C05459=1036.892,199.559,395.178,170.238,41.811,157.916
C05460=1036.886,199.310,395.204,170.234,41.811,157.916
C05461=1036.880,199.061,395.228,170.231,41.811,157.916
C05462=1036.873,198.813,395.253,170.228,41.811,157.916
C05463=1036.868,198.564,395.277,170.225,41.811,157.916
C05464=1036.861,198.316,395.302,170.222,41.811,157.915
C05465=1036.855,198.066,395.327,170.219,41.810,157.915
C05466=1036.848,197.818,395.351,170.215,41.810,157.915
C05467=1036.843,197.570,395.376,170.212,41.810,157.915
C05468=1036.836,197.321,395.400,170.209,41.810,157.915
C05469=1036.830,197.072,395.425,170.206,41.810,157.914
C05470=1036.824,196.823,395.450,170.203,41.810,157.914
C05471=1036.817,196.575,395.474,170.199,41.810,157.914
C05472=1036.812,196.326,395.499,170.196,41.810,157.914
C05473=1036.805,196.077,395.523,170.193,41.809,157.913
C05474=1036.799,195.828,395.548,170.190,41.810,157.913
C05475=1036.793,195.580,395.572,170.187,41.810,157.913
C05476=1036.787,195.331,395.597,170.184,41.809,157.913
C05477=1036.780,195.082,395.621,170.180,41.809,157.913
C05478=1036.774,194.833,395.646,170.177,41.809,157.912
C05479=1036.768,194.585,395.670,170.174,41.809,157.912
C05480=1036.762,194.336,395.695,170.172,41.809,157.912
C05481=1036.755,194.087,395.719,170.169,41.809,157.912
C05482=1036.749,193.839,395.744,170.165,41.809,157.912
C05483=1036.743,193.590,395.768,170.162,41.808,157.911
C05484=1036.737,193.341,395.792,170.159,41.809,157.911
C05485=1036.731,193.092,395.816,170.156,41.809,157.911
C05486=1036.725,192.844,395.841,170.153,41.808,157.911
C05487=1036.718,192.595,395.865,170.150,41.808,157.910
C05488=1036.713,192.346,395.890,170.147,41.809,157.910
C05489=1036.706,192.097,395.914,170.144,41.808,157.910
C05490=1036.701,191.849,395.939,170.141,41.808,157.910
C05491=1036.694,191.600,395.963,170.138,41.808,157.910
C05492=1036.688,191.351,395.987,170.135,41.808,157.910
C05493=1036.682,191.103,396.011,170.132,41.808,157.909
C05494=1036.676,190.853,396.036,170.128,41.808,157.909
C05495=1036.670,190.606,396.060,170.125,41.808,157.909
C05496=1036.664,190.356,396.085,170.122,41.808,157.909
C05497=1036.657,190.107,396.109,170.120,41.808,157.909
C05498=1036.652,189.859,396.133,170.117,41.807,157.908
C05499=1036.645,189.610,396.157,170.114,41.807,157.908
C05500=1036.639,189.326,396.185,170.110,41.807,157.908
C05501=1036.632,189.041,396.213,170.106,41.808,157.908
C05502=1036.625,188.758,396.240,170.103,41.807,157.907
C05503=1036.618,188.473,396.268,170.100,41.807,157.907
C05504=1036.612,188.225,396.292,170.097,41.807,157.907
C05505=1036.606,187.976,396.317,170.094,41.807,157.907
C05506=1036.600,187.728,396.340,170.091,41.807,157.907
C05507=1036.594,187.478,396.365,170.088,41.807,157.906
C05508=1036.588,187.230,396.389,170.085,41.807,157.906
C05509=1036.582,186.981,396.413,170.082,41.807,157.906
C05510=1036.576,186.732,396.437,170.079,41.807,157.906
C05511=1036.570,186.483,396.461,170.075,41.807,157.906
C05512=1036.564,186.235,396.485,170.073,41.807,157.906
C05513=1036.558,185.986,396.509,170.070,41.807,157.905
C05514=1036.552,185.737,396.533,170.067,41.806,157.905
C05515=1036.546,185.488,396.557,170.064,41.806,157.905
C05516=1036.541,185.239,396.581,170.062,41.806,157.905
C05517=1036.535,184.991,396.605,170.059,41.806,157.905
C05518=1036.529,184.742,396.629,170.055,41.806,157.904
C05519=1036.523,184.493,396.653,170.052,41.806,157.904
C05520=1036.517,184.244,396.678,170.049,41.806,157.904
C05521=1036.511,183.996,396.701,170.047,41.806,157.904
C05522=1036.505,183.746,396.726,170.044,41.806,157.904
C05523=1036.499,183.498,396.750,170.041,41.806,157.903
C05524=1036.493,183.250,396.773,170.037,41.806,157.903
C05525=1036.486,183.000,396.796,170.035,41.806,157.903
C05526=1036.480,182.752,396.820,170.032,41.807,157.903
C05527=1036.474,182.503,396.844,170.029,41.806,157.903
C05528=1036.468,182.254,396.867,170.026,41.807,157.903
C05529=1036.461,182.005,396.891,170.023,41.807,157.903
C05530=1036.455,181.757,396.915,170.020,41.807,157.902
C05531=1036.449,181.507,396.938,170.018,41.807,157.902
C05532=1036.442,181.259,396.961,170.015,41.807,157.902
C05533=1036.436,181.010,396.985,170.012,41.807,157.902
C05534=1036.430,180.761,397.008,170.009,41.808,157.902
C05535=1036.423,180.512,397.032,170.005,41.808,157.902
C05536=1036.418,180.264,397.055,170.002,41.808,157.902
C05537=1036.411,180.015,397.079,170.000,41.808,157.901
C05538=1036.405,179.766,397.102,169.997,41.808,157.901
C05539=1036.399,179.517,397.126,169.994,41.809,157.901
C05540=1036.393,179.268,397.149,169.991,41.809,157.901
C05541=1036.386,179.020,397.172,169.988,41.809,157.901
C05542=1036.380,178.770,397.195,169.986,41.809,157.901
C05543=1036.374,178.522,397.219,169.983,41.810,157.901
C05544=1036.367,178.272,397.242,169.979,41.809,157.900
C05545=1036.361,178.024,397.266,169.976,41.810,157.900
C05546=1036.356,177.775,397.289,169.974,41.810,157.900
C05547=1036.349,177.526,397.313,169.971,41.810,157.900
C05548=1036.342,177.278,397.335,169.968,41.810,157.900
C05549=1036.336,177.029,397.359,169.965,41.811,157.900
C05550=1036.330,176.780,397.382,169.963,41.810,157.900
C05551=1036.324,176.531,397.406,169.960,41.811,157.899
C05552=1036.318,176.282,397.429,169.957,41.811,157.899
C05553=1036.312,176.033,397.452,169.954,41.811,157.899
C05554=1036.306,175.785,397.476,169.952,41.811,157.899
C05555=1036.299,175.535,397.499,169.949,41.812,157.899
C05556=1036.293,175.287,397.522,169.946,41.812,157.899
C05557=1036.287,175.038,397.545,169.942,41.812,157.899
C05558=1036.281,174.789,397.569,169.940,41.812,157.899
C05559=1036.275,174.540,397.592,169.937,41.813,157.898
C05560=1036.269,174.291,397.615,169.934,41.812,157.898
C05561=1036.263,174.043,397.638,169.931,41.813,157.898
C05562=1036.256,173.794,397.662,169.929,41.813,157.898
C05563=1036.250,173.545,397.685,169.926,41.813,157.898
C05564=1036.244,173.261,397.712,169.923,41.813,157.898
C05565=1036.236,172.976,397.738,169.920,41.814,157.898
C05566=1036.230,172.692,397.765,169.916,41.813,157.897
C05567=1036.222,172.406,397.791,169.913,41.814,157.897
C05568=1036.216,172.158,397.814,169.910,41.814,157.897
C05569=1036.211,171.909,397.837,169.907,41.814,157.897
C05570=1036.204,171.661,397.860,169.904,41.814,157.897
C05571=1036.198,171.411,397.883,169.902,41.815,157.897
C05572=1036.192,171.162,397.906,169.899,41.815,157.897
C05573=1036.186,170.914,397.930,169.896,41.815,157.896
C05574=1036.180,170.665,397.952,169.894,41.815,157.896
C05575=1036.174,170.415,397.976,169.891,41.816,157.896
C05576=1036.167,170.167,397.998,169.888,41.816,157.896
C05577=1036.162,169.918,398.021,169.886,41.816,157.896
C05578=1036.156,169.670,398.045,169.883,41.816,157.896
C05579=1036.150,169.421,398.068,169.879,41.817,157.896
C05580=1036.144,169.171,398.091,169.877,41.816,157.895
C05581=1036.137,168.923,398.113,169.874,41.817,157.895
C05582=1036.131,168.674,398.136,169.871,41.817,157.895
C05583=1036.126,168.425,398.159,169.869,41.817,157.895
C05584=1036.120,168.176,398.183,169.866,41.817,157.895
C05585=1036.114,167.928,398.206,169.863,41.818,157.895
C05586=1036.107,167.679,398.228,169.861,41.818,157.895
C05587=1036.101,167.429,398.251,169.858,41.818,157.895
C05588=1036.095,167.180,398.274,169.856,41.818,157.895
C05589=1036.090,166.932,398.297,169.853,41.818,157.894
C05590=1036.084,166.683,398.320,169.850,41.819,157.894
C05591=1036.077,166.434,398.343,169.847,41.818,157.894
C05592=1036.072,166.185,398.366,169.844,41.819,157.894
C05593=1036.066,165.936,398.389,169.841,41.819,157.894
C05594=1036.060,165.687,398.412,169.839,41.819,157.894
C05595=1036.055,165.439,398.434,169.836,41.819,157.894
C05596=1036.047,165.189,398.457,169.834,41.820,157.894
C05597=1036.042,164.940,398.480,169.831,41.820,157.893
C05598=1036.036,164.691,398.503,169.828,41.820,157.893
C05599=1036.030,164.443,398.526,169.826,41.820,157.893
C05600=1036.024,164.194,398.548,169.823,41.820,157.893
C05601=1036.018,163.945,398.571,169.821,41.821,157.893
C05602=1036.012,163.696,398.594,169.818,41.821,157.893
C05603=1036.007,163.447,398.617,169.814,41.821,157.893
C05604=1036.001,163.198,398.640,169.812,41.821,157.893
C05605=1035.994,162.950,398.663,169.809,41.822,157.892
C05606=1035.989,162.701,398.685,169.807,41.822,157.892
C05607=1035.983,162.452,398.708,169.804,41.822,157.892
C05608=1035.977,162.203,398.731,169.801,41.822,157.892
C05609=1035.971,161.955,398.754,169.799,41.822,157.892
C05610=1035.965,161.706,398.777,169.796,41.823,157.892
C05611=1035.960,161.456,398.799,169.794,41.822,157.892
C05612=1035.954,161.207,398.822,169.791,41.823,157.892
C05613=1035.947,160.959,398.844,169.789,41.823,157.891
C05614=1035.942,160.710,398.867,169.786,41.824,157.891
C05615=1035.936,160.461,398.890,169.784,41.823,157.891
C05616=1035.930,160.212,398.913,169.780,41.824,157.891
C05617=1035.925,159.962,398.935,169.777,41.824,157.891
C05618=1035.918,159.714,398.958,169.775,41.824,157.891
C05619=1035.912,159.465,398.980,169.772,41.825,157.891
C05620=1035.906,159.216,399.003,169.770,41.825,157.891
C05621=1035.900,158.967,399.025,169.767,41.825,157.891
C05622=1035.893,158.719,399.047,169.764,41.826,157.891
C05623=1035.888,158.470,399.070,169.762,41.826,157.890
C05624=1035.882,158.220,399.091,169.759,41.827,157.890
C05625=1035.875,157.972,399.114,169.757,41.827,157.890
C05626=1035.870,157.722,399.136,169.754,41.827,157.890
C05627=1035.863,157.474,399.158,169.751,41.828,157.890
C05628=1035.856,157.189,399.184,169.748,41.828,157.890
C05629=1035.849,156.904,399.209,169.745,41.829,157.890
C05630=1035.842,156.618,399.235,169.743,41.829,157.890
C05631=1035.835,156.333,399.260,169.740,41.829,157.890
C05632=1035.829,156.085,399.283,169.737,41.830,157.890
C05633=1035.823,155.835,399.305,169.734,41.830,157.889
C05634=1035.817,155.587,399.327,169.732,41.830,157.889
C05635=1035.811,155.337,399.349,169.729,41.831,157.889
C05636=1035.805,155.088,399.372,169.727,41.831,157.889
C05637=1035.799,154.839,399.394,169.724,41.831,157.889
C05638=1035.792,154.591,399.416,169.722,41.832,157.889
C05639=1035.786,154.342,399.439,169.719,41.832,157.889
C05640=1035.780,154.093,399.460,169.717,41.832,157.889
C05641=1035.775,153.844,399.482,169.714,41.833,157.889
C05642=1035.768,153.596,399.504,169.711,41.833,157.889
C05643=1035.763,153.346,399.526,169.709,41.834,157.889
C05644=1035.756,153.097,399.549,169.706,41.834,157.889
C05645=1035.750,152.848,399.570,169.704,41.834,157.888
C05646=1035.744,152.600,399.593,169.700,41.835,157.888
C05647=1035.738,152.350,399.614,169.698,41.835,157.888
C05648=1035.732,152.101,399.637,169.695,41.835,157.888
C05649=1035.726,151.852,399.659,169.692,41.836,157.888
C05650=1035.720,151.603,399.681,169.690,41.836,157.888
C05651=1035.713,151.355,399.703,169.687,41.837,157.888
C05652=1035.707,151.105,399.725,169.685,41.837,157.888
C05653=1035.701,150.857,399.746,169.682,41.837,157.888
C05654=1035.696,150.608,399.769,169.680,41.838,157.888
C05655=1035.689,150.359,399.790,169.677,41.839,157.888
C05656=1035.683,150.109,399.812,169.675,41.839,157.888
C05657=1035.677,149.861,399.834,169.672,41.839,157.888
C05658=1035.671,149.612,399.856,169.670,41.840,157.887
C05659=1035.664,149.362,399.878,169.667,41.840,157.887
C05660=1035.658,149.114,399.900,169.665,41.840,157.887
C05661=1035.653,148.865,399.922,169.662,41.841,157.887
C05662=1035.647,148.616,399.943,169.660,41.841,157.887
C05663=1035.641,148.367,399.965,169.657,41.841,157.887
C05664=1035.634,148.118,399.987,169.655,41.842,157.887
C05665=1035.628,147.869,400.009,169.652,41.842,157.887
C05666=1035.622,147.620,400.031,169.650,41.842,157.887
C05667=1035.616,147.371,400.052,169.647,41.843,157.887
C05668=1035.610,147.122,400.074,169.644,41.844,157.887
C05669=1035.604,146.873,400.096,169.642,41.844,157.887
C05670=1035.598,146.624,400.118,169.639,41.845,157.887
C05671=1035.592,146.375,400.139,169.637,41.845,157.886
C05672=1035.585,146.126,400.161,169.634,41.845,157.886
C05673=1035.580,145.877,400.182,169.632,41.846,157.886
C05674=1035.574,145.628,400.204,169.629,41.847,157.886
C05675=1035.567,145.379,400.225,169.627,41.847,157.886
C05676=1035.561,145.130,400.247,169.624,41.847,157.886
C05677=1035.555,144.881,400.269,169.622,41.848,157.886
C05678=1035.549,144.632,400.291,169.619,41.848,157.886
C05679=1035.543,144.383,400.312,169.617,41.849,157.886
C05680=1035.537,144.134,400.334,169.614,41.849,157.886
C05681=1035.530,143.885,400.355,169.612,41.850,157.886
C05682=1035.524,143.636,400.377,169.609,41.850,157.886
C05683=1035.518,143.388,400.398,169.607,41.850,157.886
C05684=1035.512,143.138,400.420,169.604,41.851,157.886
C05685=1035.506,142.889,400.441,169.602,41.852,157.886
C05686=1035.500,142.640,400.463,169.599,41.852,157.886
C05687=1035.494,142.391,400.484,169.597,41.852,157.886
C05688=1035.488,142.142,400.506,169.594,41.853,157.885
C05689=1035.482,141.893,400.527,169.592,41.853,157.885
C05690=1035.476,141.644,400.549,169.589,41.854,157.885
C05691=1035.469,141.395,400.570,169.587,41.854,157.885
C05692=1035.462,141.110,400.595,169.584,41.855,157.885
C05693=1035.456,140.824,400.619,169.581,41.855,157.885
C05694=1035.449,140.539,400.644,169.578,41.856,157.885
C05695=1035.442,140.254,400.669,169.576,41.857,157.885
C05696=1035.436,140.005,400.690,169.573,41.857,157.885
C05697=1035.430,139.755,400.711,169.571,41.857,157.885
C05698=1035.423,139.506,400.732,169.568,41.858,157.885
C05699=1035.418,139.258,400.753,169.566,41.858,157.885
C05700=1035.412,139.009,400.775,169.563,41.859,157.885
C05701=1035.405,138.759,400.797,169.561,41.859,157.885
C05702=1035.399,138.510,400.818,169.558,41.860,157.885
C05703=1035.393,138.262,400.839,169.556,41.860,157.885
C05704=1035.387,138.012,400.860,169.553,41.861,157.885
C05705=1035.381,137.763,400.882,169.551,41.861,157.884
C05706=1035.375,137.515,400.902,169.548,41.862,157.884
C05707=1035.368,137.266,400.924,169.546,41.862,157.884
C05708=1035.362,137.016,400.946,169.543,41.863,157.884
C05709=1035.357,136.767,400.966,169.541,41.864,157.884
C05710=1035.350,136.518,400.987,169.539,41.864,157.884
C05711=1035.344,136.269,401.009,169.536,41.865,157.884
C05712=1035.338,136.021,401.030,169.534,41.865,157.884
C05713=1035.332,135.771,401.050,169.531,41.866,157.884
C05714=1035.326,135.522,401.072,169.529,41.866,157.884
C05715=1035.320,135.273,401.093,169.526,41.867,157.884
C05716=1035.313,135.025,401.114,169.524,41.867,157.884
C05717=1035.307,134.775,401.135,169.521,41.868,157.884
C05718=1035.301,134.527,401.156,169.520,41.869,157.884
C05719=1035.295,134.277,401.178,169.516,41.869,157.884
C05720=1035.289,134.027,401.198,169.514,41.869,157.884
C05721=1035.283,133.779,401.219,169.513,41.870,157.884
C05722=1035.277,133.530,401.241,169.510,41.871,157.884
C05723=1035.271,133.280,401.262,169.508,41.871,157.884
C05724=1035.264,133.032,401.282,169.505,41.871,157.884
C05725=1035.258,132.783,401.304,169.503,41.872,157.884
C05726=1035.252,132.534,401.324,169.500,41.873,157.883
C05727=1035.246,132.285,401.346,169.498,41.873,157.883
C05728=1035.240,132.035,401.366,169.496,41.874,157.883
C05729=1035.234,131.787,401.387,169.493,41.874,157.883
C05730=1035.228,131.538,401.409,169.491,41.875,157.883
C05731=1035.222,131.289,401.429,169.488,41.875,157.883
C05732=1035.216,131.040,401.450,169.486,41.876,157.883
C05733=1035.210,130.790,401.471,169.483,41.876,157.883
C05734=1035.203,130.542,401.492,169.481,41.877,157.883
C05735=1035.197,130.292,401.512,169.478,41.878,157.883
C05736=1035.191,130.044,401.534,169.476,41.878,157.883
C05737=1035.185,129.794,401.554,169.474,41.879,157.883
C05738=1035.178,129.545,401.575,169.471,41.879,157.883
C05739=1035.172,129.296,401.596,169.469,41.880,157.883
C05740=1035.166,129.047,401.617,169.466,41.881,157.883
C05741=1035.160,128.798,401.637,169.464,41.882,157.883
C05742=1035.154,128.549,401.657,169.461,41.882,157.883
C05743=1035.147,128.300,401.678,169.459,41.882,157.883
C05744=1035.141,128.051,401.698,169.456,41.883,157.883
C05745=1035.135,127.802,401.720,169.454,41.884,157.883
C05746=1035.129,127.553,401.740,169.451,41.885,157.883
C05747=1035.122,127.303,401.760,169.449,41.885,157.883
C05748=1035.116,127.055,401.781,169.448,41.886,157.883
C05749=1035.110,126.805,401.802,169.445,41.886,157.883
C05750=1035.103,126.556,401.822,169.442,41.887,157.883
C05751=1035.097,126.308,401.843,169.440,41.888,157.883
C05752=1035.091,126.058,401.864,169.438,41.888,157.883
C05753=1035.085,125.809,401.884,169.435,41.889,157.883
C05754=1035.078,125.560,401.905,169.433,41.889,157.883
C05755=1035.073,125.311,401.925,169.431,41.890,157.883
C05756=1035.065,125.026,401.948,169.428,41.891,157.883
C05757=1035.058,124.740,401.972,169.425,41.892,157.883
C05758=1035.051,124.454,401.996,169.422,41.892,157.882
C05759=1035.044,124.169,402.020,169.420,41.893,157.883
C05760=1035.038,123.920,402.040,169.417,41.894,157.882
C05761=1035.032,123.670,402.061,169.415,41.894,157.882
C05762=1035.026,123.421,402.081,169.412,41.895,157.882
C05763=1035.019,123.173,402.102,169.410,41.895,157.882
C05764=1035.014,122.923,402.122,169.407,41.896,157.882
C05765=1035.008,122.675,402.142,169.405,41.897,157.882
C05766=1035.001,122.425,402.163,169.403,41.897,157.882
C05767=1034.995,122.177,402.183,169.400,41.898,157.882
C05768=1034.989,121.927,402.204,169.398,41.898,157.882
C05769=1034.983,121.678,402.224,169.397,41.899,157.882
C05770=1034.976,121.429,402.244,169.393,41.900,157.882
C05771=1034.970,121.180,402.264,169.392,41.900,157.882
C05772=1034.964,120.931,402.286,169.389,41.901,157.882
C05773=1034.958,120.682,402.306,169.387,41.901,157.882
C05774=1034.952,120.432,402.326,169.385,41.902,157.882
C05775=1034.946,120.183,402.347,169.382,41.903,157.882
C05776=1034.940,119.935,402.367,169.380,41.903,157.882
C05777=1034.934,119.685,402.387,169.377,41.904,157.882
C05778=1034.928,119.436,402.407,169.375,41.904,157.882
C05779=1034.922,119.187,402.429,169.373,41.905,157.882
C05780=1034.916,118.938,402.449,169.370,41.906,157.882
C05781=1034.910,118.689,402.469,169.368,41.906,157.882
C05782=1034.903,118.440,402.489,169.366,41.907,157.882
C05783=1034.898,118.191,402.510,169.363,41.907,157.882
C05784=1034.891,117.941,402.530,169.361,41.908,157.882
C05785=1034.885,117.692,402.550,169.359,41.908,157.882
C05786=1034.879,117.444,402.570,169.356,41.909,157.882
C05787=1034.873,117.194,402.591,169.354,41.910,157.882
C05788=1034.867,116.945,402.611,169.351,41.910,157.882
C05789=1034.861,116.697,402.631,169.349,41.911,157.882
C05790=1034.854,116.447,402.652,169.347,41.911,157.882
C05791=1034.849,116.198,402.672,169.344,41.912,157.881
C05792=1034.843,115.949,402.692,169.342,41.913,157.882
C05793=1034.837,115.700,402.712,169.340,41.913,157.881
C05794=1034.831,115.451,402.732,169.338,41.914,157.882
C05795=1034.825,115.202,402.753,169.335,41.914,157.881
C05796=1034.819,114.952,402.773,169.333,41.915,157.881
C05797=1034.813,114.704,402.793,169.331,41.916,157.881
C05798=1034.807,114.455,402.813,169.329,41.916,157.881
C05799=1034.800,114.205,402.834,169.327,41.916,157.881
C05800=1034.795,113.956,402.854,169.324,41.917,157.881
C05801=1034.789,113.707,402.874,169.322,41.918,157.881
C05802=1034.783,113.457,402.894,169.320,41.918,157.881
C05803=1034.777,113.208,402.914,169.317,41.919,157.881
C05804=1034.771,112.959,402.934,169.315,41.919,157.881
C05805=1034.764,112.710,402.954,169.313,41.920,157.881
C05806=1034.758,112.461,402.974,169.310,41.921,157.881
C05807=1034.752,112.212,402.994,169.308,41.922,157.881
C05808=1034.745,111.963,403.014,169.306,41.922,157.881
C05809=1034.739,111.714,403.034,169.303,41.923,157.881
C05810=1034.734,111.465,403.053,169.301,41.923,157.881
C05811=1034.727,111.215,403.074,169.299,41.924,157.881
C05812=1034.721,110.966,403.094,169.296,41.925,157.881
C05813=1034.715,110.717,403.114,169.294,41.925,157.881
C05814=1034.709,110.468,403.134,169.291,41.926,157.881
C05815=1034.703,110.218,403.153,169.289,41.927,157.881
C05816=1034.697,109.970,403.173,169.287,41.927,157.881
C05817=1034.691,109.721,403.193,169.285,41.928,157.881
C05818=1034.684,109.471,403.212,169.283,41.929,157.881
C05819=1034.678,109.222,403.232,169.281,41.929,157.881
C05820=1034.671,108.936,403.255,169.278,41.930,157.881
C05821=1034.664,108.651,403.277,169.275,41.931,157.881
C05822=1034.656,108.365,403.300,169.272,41.932,157.881
C05823=1034.649,108.079,403.323,169.270,41.933,157.881
C05824=1034.643,107.830,403.342,169.267,41.933,157.881
C05825=1034.637,107.581,403.362,169.265,41.934,157.881
C05826=1034.631,107.333,403.382,169.263,41.935,157.881
C05827=1034.625,107.083,403.402,169.260,41.936,157.881
C05828=1034.619,106.834,403.421,169.259,41.937,157.881
C05829=1034.612,106.585,403.441,169.256,41.937,157.881
C05830=1034.606,106.336,403.460,169.254,41.938,157.881
C05831=1034.600,106.086,403.480,169.252,41.938,157.881
C05832=1034.594,105.837,403.500,169.250,41.939,157.881
C05833=1034.588,105.588,403.520,169.247,41.940,157.881
C05834=1034.581,105.340,403.539,169.245,41.941,157.881
C05835=1034.575,105.089,403.559,169.243,41.941,157.881
C05836=1034.569,104.841,403.579,169.240,41.942,157.881
C05837=1034.563,104.592,403.599,169.238,41.942,157.881
C05838=1034.556,104.343,403.617,169.236,41.943,157.881
C05839=1034.550,104.094,403.637,169.233,41.944,157.881
C05840=1034.544,103.844,403.657,169.231,41.944,157.881
C05841=1034.538,103.595,403.677,169.229,41.945,157.881
C05842=1034.532,103.345,403.696,169.226,41.946,157.881
C05843=1034.526,103.097,403.715,169.224,41.947,157.881
C05844=1034.520,102.848,403.735,169.222,41.947,157.881
C05845=1034.513,102.598,403.755,169.220,41.948,157.881
C05846=1034.508,102.349,403.774,169.218,41.948,157.881
C05847=1034.501,102.100,403.793,169.216,41.949,157.881
C05848=1034.495,101.851,403.813,169.213,41.950,157.881
C05849=1034.489,101.602,403.833,169.211,41.951,157.881
C05850=1034.484,101.352,403.852,169.209,41.951,157.881
C05851=1034.476,101.103,403.872,169.206,41.952,157.881
C05852=1034.471,100.854,403.891,169.204,41.952,157.881
C05853=1034.465,100.605,403.911,169.202,41.953,157.881
C05854=1034.459,100.355,403.930,169.199,41.954,157.881
C05855=1034.453,100.107,403.950,169.197,41.955,157.881
C05856=1034.447,99.858,403.969,169.195,41.955,157.881
C05857=1034.440,99.607,403.988,169.192,41.956,157.881
C05858=1034.434,99.359,404.008,169.190,41.957,157.881
C05859=1034.428,99.109,404.027,169.188,41.957,157.881
C05860=1034.421,98.860,404.046,169.186,41.958,157.881
C05861=1034.415,98.612,404.066,169.184,41.959,157.881
C05862=1034.409,98.362,404.084,169.182,41.959,157.881
C05863=1034.402,98.113,404.103,169.179,41.961,157.881
C05864=1034.396,97.864,404.123,169.177,41.961,157.881
C05865=1034.390,97.615,404.142,169.175,41.962,157.881
C05866=1034.384,97.365,404.161,169.172,41.963,157.881
C05867=1034.377,97.117,404.180,169.170,41.963,157.881
C05868=1034.371,96.867,404.200,169.168,41.964,157.881
C05869=1034.365,96.618,404.218,169.165,41.965,157.881
C05870=1034.359,96.369,404.238,169.163,41.965,157.881
C05871=1034.352,96.120,404.257,169.161,41.966,157.881
C05872=1034.346,95.870,404.277,169.159,41.967,157.881
C05873=1034.340,95.621,404.295,169.157,41.968,157.881
C05874=1034.334,95.372,404.314,169.155,41.969,157.881
C05875=1034.327,95.123,404.334,169.152,41.969,157.881
C05876=1034.322,94.874,404.353,169.150,41.970,157.881
C05877=1034.315,94.625,404.372,169.148,41.971,157.881
C05878=1034.310,94.375,404.391,169.145,41.971,157.881
C05879=1034.303,94.127,404.410,169.143,41.972,157.881
C05880=1034.297,93.877,404.430,169.141,41.973,157.881
C05881=1034.291,93.628,404.448,169.138,41.974,157.881
C05882=1034.285,93.379,404.467,169.136,41.975,157.881
C05883=1034.279,93.129,404.486,169.134,41.975,157.881
C05884=1034.271,92.844,404.508,169.132,41.976,157.881
C05885=1034.264,92.557,404.530,169.129,41.977,157.881
C05886=1034.257,92.272,404.552,169.127,41.977,157.881
C05887=1034.250,91.986,404.574,169.124,41.978,157.881
C05888=1034.244,91.737,404.593,169.122,41.979,157.881
C05889=1034.238,91.488,404.612,169.119,41.980,157.880
C05890=1034.231,91.239,404.631,169.117,41.981,157.881
C05891=1034.226,90.990,404.650,169.115,41.981,157.880
C05892=1034.219,90.741,404.669,169.112,41.982,157.881
C05893=1034.214,90.491,404.688,169.110,41.982,157.880
C05894=1034.207,90.242,404.707,169.108,41.983,157.881
C05895=1034.201,89.993,404.726,169.106,41.984,157.881
C05896=1034.195,89.743,404.745,169.103,41.985,157.880
C05897=1034.189,89.494,404.763,169.102,41.986,157.881
C05898=1034.182,89.245,404.782,169.100,41.987,157.881
C05899=1034.176,88.996,404.801,169.097,41.987,157.880
C05900=1034.170,88.747,404.820,169.095,41.988,157.881
C05901=1034.164,88.497,404.838,169.093,41.989,157.881
C05902=1034.157,88.248,404.857,169.090,41.990,157.881
C05903=1034.151,87.999,404.876,169.088,41.990,157.881
C05904=1034.145,87.750,404.895,169.086,41.991,157.881
C05905=1034.139,87.501,404.914,169.083,41.992,157.881
C05906=1034.132,87.252,404.932,169.081,41.993,157.881
C05907=1034.126,87.002,404.951,169.079,41.993,157.881
C05908=1034.119,86.753,404.970,169.077,41.995,157.881
C05909=1034.113,86.504,404.988,169.075,41.995,157.881
C05910=1034.107,86.255,405.007,169.073,41.996,157.881
C05911=1034.101,86.005,405.025,169.070,41.997,157.881
C05912=1034.095,85.756,405.044,169.068,41.998,157.881
C05913=1034.088,85.507,405.063,169.066,41.998,157.881
C05914=1034.082,85.258,405.081,169.063,41.999,157.881
C05915=1034.075,85.009,405.100,169.061,42.000,157.881
C05916=1034.070,84.759,405.119,169.059,42.000,157.881
C05917=1034.063,84.510,405.138,169.056,42.001,157.881
C05918=1034.057,84.261,405.156,169.055,42.002,157.881
C05919=1034.051,84.011,405.174,169.053,42.003,157.881
C05920=1034.044,83.762,405.193,169.050,42.004,157.881
C05921=1034.038,83.513,405.212,169.048,42.005,157.881
C05922=1034.032,83.263,405.231,169.046,42.005,157.881
C05923=1034.026,83.014,405.250,169.043,42.006,157.881
C05924=1034.020,82.766,405.268,169.041,42.007,157.881
C05925=1034.014,82.516,405.286,169.039,42.007,157.881
C05926=1034.007,82.267,405.304,169.036,42.008,157.881
C05927=1034.001,82.018,405.323,169.034,42.009,157.881
C05928=1033.995,81.769,405.342,169.032,42.010,157.881
C05929=1033.989,81.519,405.360,169.029,42.011,157.881
C05930=1033.983,81.270,405.379,169.028,42.012,157.881
C05931=1033.976,81.020,405.398,169.026,42.012,157.881
C05932=1033.970,80.771,405.416,169.024,42.013,157.881
C05933=1033.964,80.522,405.434,169.021,42.014,157.881
C05934=1033.958,80.273,405.452,169.019,42.014,157.881
C05935=1033.952,80.024,405.471,169.017,42.015,157.881
C05936=1033.946,79.775,405.490,169.014,42.016,157.881
C05937=1033.940,79.525,405.508,169.012,42.017,157.881
C05938=1033.933,79.276,405.527,169.010,42.017,157.881
C05939=1033.927,79.027,405.546,169.007,42.018,157.881
C05940=1033.921,78.778,405.563,169.005,42.019,157.881
C05941=1033.915,78.529,405.582,169.004,42.020,157.881
C05942=1033.908,78.279,405.600,169.002,42.020,157.881
C05943=1033.902,78.030,405.618,168.999,42.021,157.881
C05944=1033.896,77.781,405.637,168.997,42.022,157.881
C05945=1033.890,77.531,405.656,168.995,42.022,157.881
C05946=1033.883,77.282,405.674,168.992,42.023,157.881
C05947=1033.878,77.033,405.692,168.990,42.024,157.881
C05948=1033.870,76.747,405.714,168.987,42.025,157.881
C05949=1033.863,76.462,405.734,168.985,42.026,157.881
C05950=1033.856,76.175,405.755,168.982,42.027,157.881
C05951=1033.849,75.889,405.776,168.979,42.028,157.881
C05952=1033.843,75.640,405.794,168.978,42.029,157.881
C05953=1033.837,75.390,405.812,168.976,42.030,157.881
C05954=1033.830,75.142,405.830,168.973,42.030,157.881
C05955=1033.824,74.893,405.848,168.971,42.031,157.881
C05956=1033.817,74.644,405.867,168.969,42.032,157.881
C05957=1033.811,74.394,405.885,168.966,42.033,157.881
C05958=1033.805,74.145,405.903,168.964,42.033,157.881
C05959=1033.799,73.895,405.921,168.962,42.034,157.881
C05960=1033.793,73.647,405.939,168.959,42.036,157.881
C05961=1033.786,73.397,405.957,168.957,42.036,157.881
C05962=1033.780,73.148,405.975,168.956,42.037,157.881
C05963=1033.774,72.898,405.993,168.953,42.038,157.881
C05964=1033.768,72.650,406.012,168.951,42.039,157.881
C05965=1033.762,72.400,406.030,168.949,42.039,157.881
C05966=1033.755,72.151,406.048,168.946,42.040,157.881
C05967=1033.749,71.901,406.066,168.944,42.041,157.881
C05968=1033.742,71.652,406.083,168.942,42.041,157.881
C05969=1033.736,71.403,406.102,168.939,42.042,157.881
C05970=1033.730,71.154,406.120,168.937,42.043,157.881
C05971=1033.724,70.904,406.138,168.936,42.044,157.881
C05972=1033.718,70.655,406.156,168.934,42.045,157.881
C05973=1033.712,70.406,406.174,168.931,42.046,157.881
C05974=1033.705,70.157,406.192,168.929,42.047,157.881
C05975=1033.699,69.907,406.210,168.927,42.047,157.881
C05976=1033.693,69.657,406.228,168.924,42.048,157.881
C05977=1033.687,69.409,406.246,168.922,42.049,157.881
C05978=1033.681,69.159,406.264,168.920,42.050,157.881
C05979=1033.674,68.910,406.281,168.917,42.050,157.881
C05980=1033.668,68.661,406.300,168.915,42.051,157.881
C05981=1033.662,68.412,406.318,168.914,42.052,157.881
C05982=1033.655,68.162,406.335,168.911,42.053,157.881
C05983=1033.649,67.913,406.354,168.909,42.054,157.881
C05984=1033.643,67.663,406.371,168.907,42.055,157.881
C05985=1033.636,67.415,406.388,168.904,42.056,157.881
C05986=1033.630,67.165,406.406,168.902,42.057,157.881
C05987=1033.624,66.916,406.425,168.900,42.057,157.881
C05988=1033.618,66.667,406.443,168.897,42.058,157.881
C05989=1033.611,66.417,406.460,168.895,42.059,157.881
C05990=1033.605,66.168,406.478,168.893,42.060,157.881
C05991=1033.599,65.919,406.495,168.890,42.060,157.881
C05992=1033.593,65.670,406.513,168.889,42.061,157.881
C05993=1033.587,65.420,406.531,168.887,42.062,157.881
C05994=1033.580,65.171,406.549,168.884,42.063,157.881
C05995=1033.574,64.921,406.566,168.882,42.064,157.881
C05996=1033.568,64.672,406.584,168.880,42.064,157.881
C05997=1033.561,64.423,406.602,168.877,42.066,157.881
C05998=1033.555,64.174,406.620,168.875,42.067,157.882
C05999=1033.548,63.924,406.637,168.873,42.067,157.882
C06000=1033.542,63.675,406.655,168.870,42.068,157.881
C06001=1033.537,63.426,406.673,168.869,42.069,157.882
C06002=1033.530,63.176,406.690,168.867,42.070,157.882
C06003=1033.523,62.927,406.707,168.864,42.071,157.882
C06004=1033.518,62.678,406.725,168.862,42.072,157.882
C06005=1033.511,62.428,406.742,168.859,42.073,157.882
C06006=1033.504,62.179,406.760,168.857,42.074,157.882
C06007=1033.498,61.929,406.778,168.855,42.075,157.882
C06008=1033.492,61.680,406.795,168.853,42.076,157.882
C06009=1033.485,61.431,406.812,168.851,42.076,157.882
C06010=1033.479,61.181,406.830,168.849,42.077,157.882
C06011=1033.472,60.933,406.847,168.846,42.078,157.882
C06012=1033.465,60.647,406.867,168.844,42.079,157.882
C06013=1033.457,60.360,406.886,168.841,42.080,157.882
C06014=1033.450,60.074,406.906,168.838,42.081,157.882
C06015=1033.443,59.789,406.927,168.835,42.082,157.882
C06016=1033.436,59.539,406.944,168.834,42.083,157.882
C06017=1033.431,59.290,406.961,168.832,42.084,157.882
C06018=1033.424,59.041,406.979,168.829,42.085,157.882
C06019=1033.417,58.791,406.996,168.827,42.086,157.882
C06020=1033.411,58.542,407.013,168.824,42.087,157.882
C06021=1033.405,58.293,407.031,168.822,42.088,157.882
C06022=1033.398,58.043,407.048,168.820,42.089,157.882
C06023=1033.392,57.794,407.066,168.817,42.090,157.882
C06024=1033.385,57.545,407.083,168.816,42.091,157.882
C06025=1033.379,57.296,407.100,168.814,42.092,157.882
C06026=1033.372,57.047,407.117,168.811,42.093,157.882
C06027=1033.366,56.796,407.135,168.809,42.094,157.882
C06028=1033.360,56.547,407.152,168.807,42.095,157.882
C06029=1033.353,56.298,407.169,168.804,42.095,157.882
C06030=1033.348,56.049,407.186,168.802,42.096,157.882
C06031=1033.341,55.800,407.204,168.799,42.097,157.882
C06032=1033.335,55.551,407.221,168.798,42.098,157.882
C06033=1033.329,55.301,407.239,168.796,42.099,157.883
C06034=1033.322,55.051,407.255,168.793,42.100,157.883
C06035=1033.316,54.802,407.272,168.791,42.100,157.882
C06036=1033.310,54.553,407.290,168.789,42.101,157.883
C06037=1033.303,54.304,407.307,168.786,42.102,157.883
C06038=1033.297,54.054,407.325,168.784,42.103,157.883
C06039=1033.291,53.805,407.341,168.782,42.104,157.883
C06040=1033.284,53.555,407.359,168.779,42.105,157.883
C06041=1033.278,53.307,407.376,168.778,42.106,157.883
C06042=1033.271,53.057,407.393,168.776,42.107,157.883
C06043=1033.266,52.808,407.410,168.773,42.108,157.883
C06044=1033.259,52.558,407.427,168.771,42.109,157.883
C06045=1033.253,52.309,407.444,168.769,42.110,157.883
C06046=1033.247,52.060,407.462,168.766,42.110,157.883
C06047=1033.241,51.810,407.478,168.764,42.111,157.883
C06048=1033.234,51.561,407.496,168.761,42.112,157.883
C06049=1033.228,51.312,407.513,168.760,42.113,157.883
C06050=1033.222,51.062,407.531,168.758,42.113,157.883
C06051=1033.216,50.813,407.547,168.755,42.114,157.883
C06052=1033.209,50.564,407.564,168.753,42.115,157.883
C06053=1033.203,50.315,407.582,168.751,42.116,157.883
C06054=1033.197,50.064,407.598,168.748,42.117,157.883
C06055=1033.191,49.816,407.615,168.746,42.118,157.883
C06056=1033.184,49.566,407.633,168.744,42.119,157.883
C06057=1033.178,49.317,407.650,168.741,42.120,157.883
C06058=1033.172,49.068,407.667,168.740,42.121,157.883
C06059=1033.165,48.819,407.684,168.738,42.121,157.883
C06060=1033.160,48.569,407.701,168.735,42.122,157.883
C06061=1033.153,48.319,407.718,168.733,42.123,157.883
C06062=1033.147,48.071,407.735,168.731,42.124,157.883
C06063=1033.140,47.821,407.752,168.728,42.124,157.883
C06064=1033.135,47.572,407.769,168.726,42.125,157.883
C06065=1033.129,47.322,407.786,168.724,42.126,157.883
C06066=1033.122,47.073,407.803,168.721,42.127,157.883
C06067=1033.116,46.824,407.820,168.719,42.128,157.883
C06068=1033.110,46.574,407.837,168.718,42.129,157.883
C06069=1033.104,46.325,407.854,168.715,42.130,157.883
C06070=1033.098,46.076,407.870,168.713,42.131,157.883
C06071=1033.092,45.826,407.888,168.711,42.131,157.883
C06072=1033.086,45.577,407.905,168.708,42.132,157.883
C06073=1033.080,45.328,407.921,168.706,42.133,157.883
C06074=1033.073,45.078,407.939,168.704,42.134,157.883
C06075=1033.067,44.829,407.956,168.701,42.134,157.883
C06076=1033.060,44.543,407.975,168.699,42.135,157.883
C06077=1033.053,44.257,407.994,168.696,42.136,157.883
C06078=1033.046,43.970,408.013,168.694,42.137,157.883
C06079=1033.038,43.684,408.033,168.692,42.138,157.883
C06080=1033.033,43.434,408.050,168.689,42.139,157.883
C06081=1033.027,43.185,408.067,168.687,42.140,157.883
C06082=1033.020,42.935,408.084,168.685,42.141,157.883
C06083=1033.014,42.687,408.101,168.682,42.142,157.883
C06084=1033.008,42.437,408.117,168.680,42.142,157.883
C06085=1033.001,42.187,408.133,168.677,42.143,157.883
C06086=1032.995,41.938,408.150,168.675,42.144,157.883
C06087=1032.989,41.689,408.167,168.674,42.145,157.883
C06088=1032.982,41.440,408.184,168.671,42.146,157.883
C06089=1032.976,41.190,408.200,168.669,42.147,157.883
C06090=1032.970,40.940,408.217,168.666,42.148,157.883
C06091=1032.964,40.692,408.234,168.664,42.149,157.883
C06092=1032.958,40.442,408.250,168.662,42.150,157.883
C06093=1032.951,40.192,408.267,168.659,42.151,157.883
C06094=1032.945,39.943,408.284,168.657,42.152,157.883
C06095=1032.939,39.694,408.300,168.656,42.152,157.884
C06096=1032.933,39.445,408.316,168.653,42.154,157.884
C06097=1032.926,39.195,408.334,168.651,42.154,157.883
C06098=1032.920,38.946,408.350,168.648,42.155,157.883
C06099=1032.914,38.697,408.366,168.646,42.156,157.884
C06100=1032.908,38.446,408.383,168.644,42.157,157.884
C06101=1032.901,38.198,408.400,168.641,42.158,157.884
C06102=1032.895,37.948,408.416,168.639,42.158,157.884
C06103=1032.889,37.698,408.433,168.637,42.159,157.884
C06104=1032.883,37.449,408.449,168.635,42.160,157.884
C06105=1032.877,37.200,408.466,168.633,42.161,157.884
C06106=1032.871,36.951,408.482,168.630,42.162,157.884
C06107=1032.863,36.701,408.498,168.628,42.163,157.884
C06108=1032.857,36.452,408.514,168.625,42.164,157.884
C06109=1032.851,36.203,408.531,168.623,42.165,157.884
C06110=1032.845,35.952,408.547,168.621,42.166,157.884
C06111=1032.838,35.704,408.564,168.618,42.167,157.884
C06112=1032.832,35.455,408.580,168.617,42.168,157.884
C06113=1032.825,35.205,408.596,168.614,42.169,157.884
C06114=1032.819,34.955,408.613,168.612,42.170,157.884
C06115=1032.813,34.706,408.628,168.610,42.171,157.884
C06116=1032.807,34.457,408.645,168.607,42.172,157.884
C06117=1032.800,34.207,408.661,168.605,42.173,157.884
C06118=1032.794,33.958,408.678,168.602,42.174,157.884
C06119=1032.787,33.709,408.694,168.601,42.175,157.884
C06120=1032.781,33.460,408.710,168.598,42.176,157.884
C06121=1032.775,33.210,408.727,168.596,42.177,157.884
C06122=1032.768,32.961,408.742,168.594,42.178,157.884
C06123=1032.762,32.711,408.759,168.591,42.178,157.884
C06124=1032.756,32.462,408.775,168.589,42.179,157.884
C06125=1032.750,32.213,408.791,168.586,42.180,157.884
C06126=1032.743,31.963,408.807,168.584,42.181,157.884
C06127=1032.737,31.714,408.824,168.583,42.182,157.884
C06128=1032.731,31.464,408.840,168.580,42.183,157.884
C06129=1032.725,31.215,408.856,168.578,42.184,157.884
C06130=1032.718,30.965,408.872,168.575,42.185,157.884
C06131=1032.712,30.716,408.888,168.573,42.186,157.884
C06132=1032.706,30.466,408.905,168.570,42.187,157.884
C06133=1032.700,30.217,408.921,168.568,42.188,157.884
C06134=1032.693,29.968,408.936,168.566,42.189,157.884
C06135=1032.687,29.719,408.953,168.564,42.190,157.884
C06136=1032.681,29.469,408.969,168.562,42.191,157.884
C06137=1032.674,29.220,408.985,168.559,42.192,157.885
C06138=1032.668,28.970,409.001,168.557,42.193,157.885
C06139=1032.662,28.721,409.018,168.555,42.193,157.884
C06140=1032.653,28.345,409.041,168.551,42.195,157.885
C06141=1032.643,27.969,409.066,168.547,42.196,157.885
C06142=1032.634,27.594,409.089,168.545,42.198,157.885
C06143=1032.624,27.219,409.113,168.541,42.199,157.885
C06144=1032.618,26.970,409.130,168.538,42.200,157.885
C06145=1032.612,26.720,409.146,168.536,42.201,157.885
C06146=1032.605,26.470,409.161,168.534,42.202,157.885
C06147=1032.599,26.221,409.178,168.531,42.203,157.885
C06148=1032.589,25.811,409.204,168.528,42.205,157.885
C06149=1032.578,25.401,409.230,168.524,42.206,157.885
C06150=1032.567,24.992,409.256,168.520,42.208,157.885
C06151=1032.557,24.582,409.281,168.516,42.210,157.885
C06152=1032.551,24.333,409.297,168.513,42.211,157.885
C06153=1032.545,24.084,409.313,168.512,42.212,157.885
C06154=1032.539,23.835,409.329,168.510,42.213,157.885
C06155=1032.532,23.584,409.345,168.507,42.214,157.885
C06156=1032.526,23.335,409.361,168.505,42.215,157.885
C06157=1032.519,23.086,409.377,168.502,42.216,157.885
C06158=1032.513,22.837,409.392,168.500,42.217,157.885
C06159=1032.507,22.587,409.408,168.497,42.218,157.885
C06160=1032.500,22.338,409.423,168.495,42.218,157.885
C06161=1032.494,22.089,409.440,168.493,42.219,157.885
C06162=1032.488,21.839,409.455,168.491,42.220,157.885
C06163=1032.482,21.590,409.471,168.488,42.221,157.885
C06164=1032.475,21.340,409.486,168.486,42.222,157.885
C06165=1032.470,21.091,409.502,168.483,42.223,157.885
C06166=1032.463,20.841,409.518,168.481,42.224,157.885
C06167=1032.457,20.592,409.534,168.479,42.225,157.885
C06168=1032.451,20.342,409.549,168.477,42.226,157.885
C06169=1032.444,20.092,409.566,168.475,42.227,157.886
C06170=1032.437,19.843,409.581,168.472,42.228,157.886
C06171=1032.432,19.593,409.597,168.470,42.229,157.886
C06172=1032.425,19.344,409.612,168.467,42.230,157.886
C06173=1032.419,19.095,409.627,168.465,42.231,157.886
C06174=1032.413,18.845,409.644,168.462,42.232,157.886
C06175=1032.406,18.596,409.659,168.460,42.233,157.886
C06176=1032.400,18.347,409.674,168.458,42.234,157.886
C06177=1032.394,18.097,409.690,168.456,42.235,157.886
C06178=1032.387,17.848,409.705,168.453,42.236,157.886
C06179=1032.381,17.599,409.721,168.451,42.237,157.886
C06180=1032.374,17.349,409.736,168.448,42.238,157.886
C06181=1032.368,17.100,409.752,168.446,42.239,157.886
C06182=1032.362,16.850,409.767,168.443,42.240,157.886
C06183=1032.355,16.601,409.783,168.442,42.241,157.886
C06184=1032.349,16.351,409.798,168.439,42.242,157.886
C06185=1032.343,16.102,409.814,168.437,42.243,157.886
C06186=1032.336,15.852,409.829,168.434,42.244,157.886
C06187=1032.331,15.602,409.845,168.432,42.245,157.886
C06188=1032.324,15.353,409.860,168.429,42.246,157.886
C06189=1032.318,15.104,409.875,168.427,42.247,157.886
C06190=1032.312,14.854,409.891,168.425,42.248,157.886
C06191=1032.305,14.605,409.906,168.423,42.249,157.886
C06192=1032.299,14.356,409.922,168.420,42.250,157.886
C06193=1032.293,14.106,409.938,168.418,42.251,157.886
C06194=1032.287,13.857,409.952,168.415,42.252,157.886
C06195=1032.281,13.608,409.968,168.413,42.253,157.886
C06196=1032.274,13.358,409.983,168.410,42.254,157.886
C06197=1032.268,13.108,409.998,168.409,42.255,157.886
C06198=1032.261,12.859,410.013,168.406,42.257,157.886
C06199=1032.255,12.610,410.028,168.404,42.257,157.886
C06200=1032.247,12.324,410.046,168.401,42.259,157.886
C06201=1032.240,12.039,410.064,168.398,42.260,157.887
C06202=1032.233,11.754,410.080,168.396,42.261,157.887
C06203=1032.225,11.469,410.098,168.393,42.263,157.887
C06204=1032.219,11.219,410.113,168.391,42.264,157.887
C06205=1032.212,10.970,410.129,168.388,42.265,157.887
C06206=1032.206,10.720,410.144,168.385,42.266,157.887
C06207=1032.200,10.471,410.158,168.383,42.267,157.887
C06208=1032.194,10.222,410.173,168.380,42.268,157.887
C06209=1032.187,9.973,410.189,168.379,42.269,157.887
C06210=1032.181,9.723,410.204,168.376,42.271,157.887
C06211=1032.174,9.474,410.219,168.374,42.272,157.887
C06212=1032.168,9.224,410.234,168.371,42.273,157.887
C06213=1032.162,8.974,410.248,168.369,42.274,157.887
C06214=1032.155,8.725,410.264,168.366,42.275,157.887
C06215=1032.149,8.476,410.279,168.365,42.276,157.887
C06216=1032.142,8.226,410.294,168.362,42.277,157.887
C06217=1032.136,7.977,410.309,168.359,42.278,157.887
C06218=1032.130,7.727,410.324,168.357,42.279,157.887
C06219=1032.124,7.478,410.339,168.354,42.280,157.887
C06220=1032.117,7.229,410.354,168.352,42.281,157.887
C06221=1032.111,6.979,410.369,168.349,42.282,157.887
C06222=1032.104,6.729,410.384,168.348,42.283,157.887
C06223=1032.098,6.480,410.399,168.345,42.284,157.887
C06224=1032.092,6.231,410.414,168.343,42.285,157.887
C06225=1032.086,5.981,410.429,168.340,42.286,157.887
C06226=1032.079,5.731,410.443,168.337,42.287,157.887
C06227=1032.073,5.482,410.458,168.335,42.288,157.888
C06228=1032.066,5.233,410.474,168.332,42.289,157.888
C06229=1032.060,4.983,410.489,168.331,42.290,157.888
C06230=1032.054,4.734,410.504,168.328,42.291,157.888
C06231=1032.048,4.484,410.519,168.326,42.292,157.888
C06232=1032.041,4.235,410.534,168.323,42.293,157.888
C06233=1032.035,3.985,410.548,168.321,42.294,157.888
C06234=1032.029,3.736,410.563,168.318,42.295,157.888
C06235=1032.023,3.486,410.578,168.316,42.296,157.888
C06236=1032.016,3.237,410.593,168.314,42.298,157.888
C06237=1032.010,2.987,410.608,168.311,42.299,157.888
C06238=1032.004,2.737,410.623,168.309,42.300,157.888
C06239=1031.998,2.488,410.637,168.306,42.301,157.888
C06240=1031.991,2.239,410.652,168.304,42.302,157.888
C06241=1031.985,1.989,410.667,168.301,42.303,157.888
C06242=1031.979,1.740,410.682,168.299,42.304,157.888
C06243=1031.973,1.491,410.697,168.297,42.305,157.888
C06244=1031.966,1.241,410.712,168.295,42.306,157.888
C06245=1031.960,0.991,410.727,168.292,42.307,157.888
C06246=1031.954,0.742,410.741,168.289,42.308,157.888
C06247=1031.948,0.493,410.756,168.287,42.309,157.888
C06248=1031.942,0.243,410.771,168.284,42.310,157.888
C06249=1031.935,-0.007,410.786,168.282,42.311,157.888
C06250=1031.929,-0.256,410.801,168.280,42.312,157.888
C06251=1031.923,-0.505,410.816,168.278,42.313,157.888
C06252=1031.917,-0.756,410.830,168.275,42.314,157.888
C06253=1031.911,-1.005,410.844,168.272,42.315,157.888
C06254=1031.905,-1.254,410.859,168.270,42.316,157.888
C06255=1031.898,-1.504,410.874,168.267,42.317,157.888
C06256=1031.893,-1.753,410.889,168.266,42.318,157.888
C06257=1031.886,-2.002,410.904,168.263,42.319,157.888
C06258=1031.880,-2.252,410.919,168.261,42.320,157.888
C06259=1031.874,-2.501,410.933,168.258,42.322,157.888
C06260=1031.868,-2.751,410.948,168.256,42.323,157.889
C06261=1031.862,-3.001,410.963,168.253,42.324,157.889
C06262=1031.856,-3.250,410.977,168.250,42.325,157.889
C06263=1031.849,-3.500,410.992,168.249,42.326,157.889
C06264=1031.842,-3.783,411.008,168.246,42.327,157.889
C06265=1031.835,-4.066,411.026,168.243,42.328,157.889
C06266=1031.828,-4.348,411.041,168.240,42.329,157.889
C06267=1031.821,-4.632,411.057,168.237,42.331,157.889
C06268=1031.814,-4.882,411.072,168.234,42.332,157.889
C06269=1031.808,-5.131,411.087,168.233,42.333,157.889
C06270=1031.802,-5.380,411.100,168.230,42.334,157.889
C06271=1031.795,-5.630,411.115,168.227,42.335,157.889
C06272=1031.788,-5.879,411.130,168.225,42.336,157.889
C06273=1031.783,-6.129,411.144,168.222,42.337,157.889
C06274=1031.776,-6.379,411.159,168.220,42.339,157.889
C06275=1031.769,-6.629,411.172,168.218,42.340,157.889
C06276=1031.764,-6.878,411.187,168.215,42.341,157.889
C06277=1031.757,-7.127,411.202,168.213,42.342,157.889
C06278=1031.751,-7.377,411.215,168.210,42.343,157.889
C06279=1031.745,-7.626,411.230,168.207,42.344,157.889
C06280=1031.738,-7.876,411.244,168.205,42.345,157.889
C06281=1031.732,-8.125,411.258,168.202,42.346,157.889
C06282=1031.726,-8.375,411.273,168.200,42.348,157.889
C06283=1031.720,-8.624,411.286,168.198,42.349,157.889
C06284=1031.713,-8.874,411.301,168.195,42.350,157.889
C06285=1031.706,-9.124,411.315,168.192,42.351,157.889
C06286=1031.701,-9.373,411.330,168.190,42.352,157.889
C06287=1031.694,-9.622,411.344,168.187,42.353,157.890
C06288=1031.688,-9.871,411.358,168.186,42.354,157.890
C06289=1031.682,-10.121,411.373,168.183,42.355,157.890
C06290=1031.676,-10.371,411.387,168.180,42.357,157.890
C06291=1031.669,-10.620,411.401,168.178,42.358,157.890
C06292=1031.663,-10.870,411.415,168.175,42.359,157.890
C06293=1031.656,-11.119,411.429,168.173,42.360,157.890
C06294=1031.650,-11.369,411.443,168.171,42.361,157.890
C06295=1031.644,-11.618,411.458,168.168,42.362,157.890
C06296=1031.638,-11.868,411.472,168.165,42.364,157.890
C06297=1031.632,-12.117,411.486,168.163,42.365,157.890
C06298=1031.625,-12.367,411.500,168.160,42.366,157.890
C06299=1031.620,-12.617,411.514,168.157,42.367,157.890
C06300=1031.612,-12.866,411.528,168.156,42.368,157.890
C06301=1031.607,-13.116,411.542,168.153,42.369,157.890
C06302=1031.601,-13.365,411.557,168.150,42.371,157.890
C06303=1031.594,-13.615,411.570,168.148,42.372,157.890
C06304=1031.588,-13.864,411.585,168.145,42.373,157.890
C06305=1031.582,-14.113,411.598,168.142,42.374,157.890
C06306=1031.576,-14.364,411.613,168.141,42.375,157.890
C06307=1031.570,-14.613,411.627,168.138,42.376,157.890
C06308=1031.563,-14.863,411.641,168.136,42.377,157.890
C06309=1031.557,-15.112,411.655,168.133,42.378,157.890
C06310=1031.551,-15.362,411.669,168.130,42.379,157.890
C06311=1031.545,-15.611,411.683,168.128,42.380,157.890
C06312=1031.538,-15.860,411.697,168.125,42.381,157.890
C06313=1031.532,-16.110,411.711,168.123,42.383,157.891
C06314=1031.526,-16.360,411.725,168.120,42.384,157.891
C06315=1031.519,-16.609,411.738,168.118,42.385,157.891
C06316=1031.513,-16.859,411.753,168.115,42.386,157.891
C06317=1031.507,-17.108,411.766,168.113,42.388,157.891
C06318=1031.501,-17.357,411.779,168.111,42.389,157.891
C06319=1031.495,-17.608,411.794,168.108,42.390,157.891
C06320=1031.488,-17.856,411.808,168.105,42.391,157.891
C06321=1031.481,-18.106,411.821,168.102,42.392,157.891
C06322=1031.475,-18.356,411.835,168.100,42.394,157.891
C06323=1031.469,-18.606,411.849,168.098,42.395,157.891
C06324=1031.463,-18.855,411.862,168.095,42.396,157.891
C06325=1031.456,-19.105,411.876,168.093,42.397,157.891
C06326=1031.450,-19.354,411.890,168.090,42.398,157.891
C06327=1031.444,-19.603,411.904,168.087,42.400,157.891
C06328=1031.437,-19.886,411.919,168.084,42.401,157.891
C06329=1031.430,-20.167,411.935,168.082,42.402,157.891
C06330=1031.423,-20.448,411.950,168.079,42.404,157.891
C06331=1031.416,-20.730,411.965,168.076,42.405,157.891
C06332=1031.409,-20.980,411.979,168.073,42.406,157.891
C06333=1031.403,-21.229,411.992,168.070,42.407,157.891
C06334=1031.396,-21.478,412.007,168.069,42.409,157.892
C06335=1031.391,-21.728,412.021,168.066,42.410,157.892
C06336=1031.384,-21.977,412.034,168.063,42.411,157.892
C06337=1031.378,-22.227,412.047,168.061,42.412,157.892
C06338=1031.372,-22.477,412.061,168.058,42.413,157.892
C06339=1031.366,-22.726,412.075,168.055,42.414,157.892
C06340=1031.359,-22.976,412.088,168.053,42.416,157.892
C06341=1031.354,-23.226,412.102,168.051,42.417,157.892
C06342=1031.347,-23.475,412.115,168.048,42.418,157.892
C06343=1031.341,-23.725,412.129,168.045,42.419,157.892
C06344=1031.334,-23.974,412.142,168.042,42.421,157.892
C06345=1031.329,-24.224,412.156,168.040,42.422,157.892
C06346=1031.322,-24.474,412.170,168.038,42.423,157.892
C06347=1031.316,-24.723,412.183,168.035,42.424,157.892
C06348=1031.310,-24.972,412.197,168.033,42.425,157.892
C06349=1031.304,-25.222,412.211,168.030,42.427,157.892
C06350=1031.297,-25.472,412.224,168.027,42.428,157.892
C06351=1031.291,-25.721,412.237,168.024,42.429,157.892
C06352=1031.286,-25.970,412.251,168.023,42.430,157.892
C06353=1031.279,-26.220,412.265,168.020,42.432,157.892
C06354=1031.273,-26.470,412.278,168.017,42.433,157.892
C06355=1031.266,-26.719,412.291,168.014,42.434,157.892
C06356=1031.261,-26.969,412.305,168.012,42.435,157.892
C06357=1031.254,-27.218,412.319,168.009,42.436,157.892
C06358=1031.248,-27.468,412.332,168.007,42.438,157.892
C06359=1031.242,-27.717,412.345,168.004,42.439,157.892
C06360=1031.235,-27.967,412.359,168.002,42.440,157.893
C06361=1031.229,-28.217,412.371,167.999,42.442,157.893
C06362=1031.223,-28.466,412.385,167.997,42.443,157.893
C06363=1031.217,-28.715,412.398,167.994,42.444,157.893
C06364=1031.210,-28.965,412.411,167.991,42.445,157.893
C06365=1031.203,-29.215,412.425,167.989,42.447,157.893
C06366=1031.198,-29.465,412.437,167.986,42.448,157.893
C06367=1031.191,-29.714,412.451,167.983,42.449,157.893
C06368=1031.185,-29.964,412.464,167.981,42.451,157.893
C06369=1031.178,-30.213,412.477,167.978,42.452,157.893
C06370=1031.172,-30.463,412.490,167.976,42.453,157.893
C06371=1031.166,-30.712,412.503,167.973,42.454,157.893
C06372=1031.159,-30.962,412.517,167.970,42.456,157.893
C06373=1031.153,-31.211,412.530,167.968,42.457,157.893
C06374=1031.147,-31.461,412.543,167.965,42.458,157.893
C06375=1031.141,-31.711,412.556,167.963,42.459,157.893
C06376=1031.135,-31.960,412.569,167.960,42.461,157.893
C06377=1031.129,-32.209,412.583,167.957,42.462,157.893
C06378=1031.122,-32.460,412.596,167.955,42.464,157.894
C06379=1031.116,-32.709,412.609,167.952,42.465,157.894
C06380=1031.110,-32.958,412.622,167.950,42.466,157.894
C06381=1031.104,-33.208,412.635,167.947,42.467,157.894
C06382=1031.098,-33.457,412.648,167.944,42.469,157.894
C06383=1031.091,-33.707,412.661,167.942,42.470,157.894
C06384=1031.085,-33.957,412.674,167.939,42.471,157.894
C06385=1031.079,-34.206,412.687,167.937,42.472,157.894
C06386=1031.072,-34.456,412.701,167.934,42.474,157.894
C06387=1031.066,-34.706,412.713,167.931,42.475,157.894
C06388=1031.060,-34.955,412.726,167.928,42.476,157.894
C06389=1031.054,-35.205,412.739,167.926,42.478,157.894
C06390=1031.048,-35.454,412.752,167.924,42.479,157.894
C06391=1031.041,-35.704,412.766,167.921,42.480,157.894
C06392=1031.035,-35.985,412.780,167.918,42.481,157.894
C06393=1031.029,-36.266,412.795,167.915,42.483,157.894
C06394=1031.022,-36.546,412.809,167.912,42.484,157.894
C06395=1031.014,-36.827,412.824,167.909,42.486,157.894
C06396=1031.008,-37.076,412.837,167.906,42.487,157.894
C06397=1031.002,-37.326,412.850,167.903,42.488,157.894
C06398=1030.996,-37.576,412.863,167.901,42.489,157.894
C06399=1030.990,-37.825,412.875,167.899,42.491,157.895
C06400=1030.984,-38.075,412.889,167.896,42.492,157.895
C06401=1030.977,-38.324,412.902,167.893,42.493,157.895
C06402=1030.972,-38.574,412.915,167.890,42.494,157.895
C06403=1030.965,-38.823,412.928,167.889,42.496,157.895
C06404=1030.959,-39.073,412.940,167.886,42.497,157.895
C06405=1030.953,-39.323,412.952,167.883,42.498,157.895
C06406=1030.947,-39.572,412.966,167.880,42.500,157.895
C06407=1030.941,-39.822,412.978,167.877,42.501,157.895
C06408=1030.934,-40.071,412.991,167.875,42.503,157.895
C06409=1030.927,-40.321,413.004,167.872,42.504,157.895
C06410=1030.921,-40.571,413.016,167.869,42.505,157.895
C06411=1030.914,-40.820,413.029,167.867,42.507,157.895
C06412=1030.908,-41.070,413.042,167.864,42.508,157.895
C06413=1030.903,-41.320,413.054,167.862,42.509,157.895
C06414=1030.896,-41.569,413.067,167.859,42.511,157.895
C06415=1030.890,-41.819,413.079,167.856,42.512,157.895
C06416=1030.884,-42.069,413.092,167.853,42.514,157.895
C06417=1030.878,-42.318,413.105,167.850,42.515,157.895
C06418=1030.871,-42.567,413.117,167.848,42.516,157.896
C06419=1030.865,-42.817,413.130,167.846,42.517,157.896
C06420=1030.859,-43.067,413.143,167.843,42.519,157.896
C06421=1030.853,-43.316,413.155,167.840,42.520,157.896
C06422=1030.846,-43.566,413.167,167.837,42.521,157.896
C06423=1030.840,-43.816,413.180,167.835,42.523,157.896
C06424=1030.834,-44.065,413.193,167.832,42.524,157.896
C06425=1030.827,-44.315,413.205,167.829,42.526,157.896
C06426=1030.822,-44.565,413.218,167.826,42.527,157.896
C06427=1030.816,-44.814,413.230,167.825,42.528,157.896
C06428=1030.809,-45.063,413.243,167.822,42.530,157.896
C06429=1030.803,-45.313,413.255,167.819,42.531,157.896
C06430=1030.797,-45.563,413.268,167.816,42.532,157.896
C06431=1030.791,-45.812,413.280,167.813,42.534,157.896
C06432=1030.785,-46.062,413.292,167.811,42.535,157.896
C06433=1030.779,-46.311,413.306,167.808,42.536,157.896
C06434=1030.772,-46.561,413.317,167.805,42.538,157.897
C06435=1030.766,-46.811,413.330,167.802,42.539,157.897
C06436=1030.760,-47.061,413.343,167.801,42.541,157.897
C06437=1030.754,-47.310,413.355,167.798,42.542,157.897
C06438=1030.748,-47.560,413.367,167.795,42.543,157.897
C06439=1030.742,-47.809,413.379,167.792,42.545,157.897
C06440=1030.735,-48.058,413.392,167.789,42.546,157.897
C06441=1030.730,-48.308,413.405,167.786,42.547,157.897
C06442=1030.724,-48.558,413.417,167.784,42.549,157.897
C06443=1030.717,-48.808,413.429,167.781,42.550,157.897
C06444=1030.711,-49.057,413.442,167.778,42.551,157.897
C06445=1030.705,-49.307,413.454,167.776,42.553,157.897
C06446=1030.699,-49.556,413.466,167.773,42.554,157.897
C06447=1030.693,-49.806,413.478,167.771,42.555,157.897
C06448=1030.687,-50.056,413.491,167.768,42.557,157.897
C06449=1030.681,-50.306,413.503,167.765,42.558,157.897
C06450=1030.675,-50.555,413.515,167.762,42.560,157.897
C06451=1030.669,-50.805,413.528,167.760,42.561,157.897
C06452=1030.662,-51.055,413.540,167.757,42.563,157.898
C06453=1030.656,-51.304,413.552,167.754,42.564,157.898
C06454=1030.649,-51.553,413.563,167.751,42.566,157.898
C06455=1030.644,-51.803,413.576,167.749,42.568,157.898
C06456=1030.636,-52.085,413.589,167.746,42.569,157.898
C06457=1030.629,-52.366,413.603,167.742,42.571,157.898
C06458=1030.622,-52.647,413.616,167.739,42.573,157.898
C06459=1030.614,-52.928,413.630,167.737,42.574,157.898
C06460=1030.609,-53.178,413.641,167.734,42.576,157.898
C06461=1030.603,-53.427,413.654,167.731,42.577,157.898
C06462=1030.596,-53.677,413.666,167.729,42.579,157.898
C06463=1030.590,-53.927,413.678,167.726,42.580,157.898
C06464=1030.583,-54.176,413.690,167.723,42.582,157.899
C06465=1030.578,-54.425,413.702,167.720,42.583,157.899
C06466=1030.571,-54.676,413.713,167.717,42.585,157.899
C06467=1030.565,-54.925,413.725,167.715,42.587,157.899
C06468=1030.559,-55.175,413.738,167.712,42.588,157.899
C06469=1030.552,-55.425,413.750,167.709,42.590,157.899
C06470=1030.546,-55.673,413.761,167.706,42.591,157.899
C06471=1030.540,-55.924,413.772,167.704,42.593,157.899
C06472=1030.534,-56.173,413.785,167.701,42.594,157.899
C06473=1030.527,-56.423,413.797,167.698,42.596,157.899
C06474=1030.521,-56.672,413.808,167.695,42.598,157.899
C06475=1030.515,-56.922,413.820,167.693,42.599,157.899
C06476=1030.509,-57.172,413.832,167.690,42.600,157.899
C06477=1030.502,-57.422,413.844,167.687,42.602,157.899
C06478=1030.496,-57.671,413.855,167.684,42.603,157.900
C06479=1030.490,-57.921,413.867,167.682,42.605,157.900
C06480=1030.484,-58.171,413.880,167.679,42.606,157.900
C06481=1030.478,-58.420,413.891,167.676,42.608,157.900
C06482=1030.471,-58.670,413.902,167.673,42.609,157.900
C06483=1030.465,-58.919,413.914,167.671,42.611,157.900
C06484=1030.460,-59.169,413.926,167.668,42.612,157.900
C06485=1030.453,-59.419,413.938,167.665,42.614,157.900
C06486=1030.447,-59.668,413.950,167.662,42.616,157.900
C06487=1030.440,-59.918,413.961,167.660,42.617,157.900
C06488=1030.435,-60.167,413.973,167.657,42.619,157.900
C06489=1030.428,-60.417,413.985,167.654,42.620,157.900
C06490=1030.422,-60.667,413.996,167.651,42.622,157.901
C06491=1030.416,-60.916,414.008,167.649,42.624,157.901
C06492=1030.410,-61.167,414.020,167.646,42.625,157.901
C06493=1030.404,-61.415,414.031,167.643,42.627,157.901
C06494=1030.398,-61.665,414.043,167.640,42.628,157.901
C06495=1030.391,-61.915,414.055,167.638,42.629,157.901
C06496=1030.386,-62.164,414.067,167.635,42.631,157.901
C06497=1030.380,-62.415,414.078,167.632,42.632,157.901
C06498=1030.373,-62.664,414.090,167.629,42.634,157.901
C06499=1030.367,-62.914,414.101,167.627,42.635,157.901
C06500=1030.361,-63.163,414.113,167.624,42.637,157.901
C06501=1030.356,-63.413,414.124,167.621,42.638,157.901
C06502=1030.349,-63.663,414.136,167.618,42.640,157.901
C06503=1030.343,-63.913,414.148,167.615,42.641,157.901
C06504=1030.337,-64.162,414.159,167.613,42.643,157.902
C06505=1030.330,-64.412,414.170,167.610,42.644,157.902
C06506=1030.325,-64.661,414.183,167.607,42.646,157.902
C06507=1030.319,-64.911,414.194,167.605,42.648,157.902
C06508=1030.312,-65.160,414.205,167.602,42.649,157.902
C06509=1030.306,-65.410,414.217,167.599,42.651,157.902
C06510=1030.300,-65.659,414.228,167.596,42.652,157.902
C06511=1030.294,-65.910,414.240,167.594,42.654,157.902
C06512=1030.289,-66.159,414.251,167.591,42.655,157.902
C06513=1030.282,-66.409,414.263,167.588,42.657,157.902
C06514=1030.276,-66.658,414.274,167.585,42.658,157.902
C06515=1030.270,-66.908,414.286,167.582,42.660,157.902
C06516=1030.264,-67.158,414.298,167.580,42.661,157.902
C06517=1030.258,-67.408,414.309,167.577,42.663,157.902
C06518=1030.252,-67.657,414.320,167.574,42.664,157.903
C06519=1030.246,-67.907,414.331,167.571,42.666,157.903
C06520=1030.239,-68.190,414.344,167.568,42.668,157.903
C06521=1030.232,-68.472,414.358,167.565,42.669,157.903
C06522=1030.226,-68.754,414.371,167.561,42.671,157.903
C06523=1030.219,-69.036,414.383,167.558,42.672,157.903
C06524=1030.213,-69.286,414.395,167.556,42.674,157.903
C06525=1030.207,-69.536,414.406,167.553,42.675,157.903
C06526=1030.201,-69.785,414.417,167.550,42.677,157.903
C06527=1030.195,-70.035,414.429,167.547,42.678,157.903
C06528=1030.189,-70.284,414.440,167.545,42.680,157.903
C06529=1030.183,-70.534,414.452,167.542,42.681,157.903
C06530=1030.177,-70.784,414.463,167.539,42.683,157.903
C06531=1030.171,-71.034,414.474,167.536,42.685,157.903
C06532=1030.165,-71.284,414.485,167.534,42.686,157.903
C06533=1030.159,-71.532,414.497,167.531,42.688,157.904
C06534=1030.153,-71.783,414.508,167.528,42.689,157.904
C06535=1030.148,-72.032,414.519,167.525,42.691,157.904
C06536=1030.142,-72.282,414.530,167.523,42.692,157.904
C06537=1030.136,-72.532,414.541,167.520,42.694,157.904
C06538=1030.130,-72.781,414.553,167.517,42.695,157.904
C06539=1030.124,-73.031,414.564,167.514,42.697,157.904
C06540=1030.118,-73.281,414.575,167.511,42.698,157.904
C06541=1030.112,-73.530,414.586,167.509,42.700,157.904
C06542=1030.106,-73.781,414.598,167.506,42.701,157.904
C06543=1030.100,-74.029,414.610,167.503,42.703,157.904
C06544=1030.095,-74.279,414.620,167.500,42.705,157.904
C06545=1030.088,-74.529,414.632,167.497,42.706,157.904
C06546=1030.083,-74.779,414.643,167.494,42.708,157.904
C06547=1030.076,-75.029,414.653,167.491,42.710,157.904
C06548=1030.070,-75.278,414.664,167.489,42.711,157.905
C06549=1030.064,-75.527,414.675,167.486,42.712,157.905
C06550=1030.058,-75.778,414.686,167.483,42.714,157.905
C06551=1030.052,-76.027,414.697,167.480,42.716,157.905
C06552=1030.046,-76.277,414.708,167.478,42.717,157.905
C06553=1030.040,-76.527,414.719,167.475,42.719,157.905
C06554=1030.033,-76.776,414.729,167.472,42.721,157.905
C06555=1030.028,-77.026,414.740,167.469,42.723,157.905
C06556=1030.021,-77.276,414.752,167.466,42.724,157.905
C06557=1030.016,-77.525,414.762,167.463,42.726,157.905
C06558=1030.010,-77.775,414.773,167.460,42.728,157.905
C06559=1030.004,-78.024,414.784,167.458,42.730,157.906
C06560=1029.998,-78.274,414.795,167.455,42.731,157.906
C06561=1029.992,-78.524,414.806,167.452,42.732,157.906
C06562=1029.986,-78.773,414.817,167.449,42.734,157.906
C06563=1029.979,-79.023,414.828,167.447,42.735,157.906
C06564=1029.974,-79.273,414.838,167.444,42.737,157.906
C06565=1029.968,-79.523,414.849,167.440,42.739,157.906
C06566=1029.962,-79.773,414.860,167.438,42.741,157.906
C06567=1029.956,-80.023,414.871,167.435,42.742,157.906
C06568=1029.949,-80.272,414.881,167.432,42.744,157.906
C06569=1029.944,-80.521,414.892,167.429,42.746,157.906
C06570=1029.937,-80.772,414.902,167.427,42.748,157.906
C06571=1029.931,-81.021,414.913,167.424,42.750,157.907
C06572=1029.925,-81.271,414.924,167.420,42.752,157.907
C06573=1029.919,-81.520,414.934,167.418,42.753,157.907
C06574=1029.913,-81.771,414.945,167.415,42.755,157.907
C06575=1029.906,-82.020,414.955,167.412,42.757,157.907
C06576=1029.901,-82.269,414.966,167.409,42.758,157.907
C06577=1029.895,-82.519,414.977,167.407,42.760,157.907
C06578=1029.888,-82.769,414.987,167.404,42.762,157.907
C06579=1029.882,-83.019,414.998,167.400,42.764,157.907
C06580=1029.876,-83.268,415.008,167.398,42.766,157.908
C06581=1029.871,-83.518,415.018,167.395,42.767,157.908
C06582=1029.864,-83.768,415.029,167.392,42.769,157.908
C06583=1029.858,-84.017,415.039,167.390,42.771,157.908
C06584=1029.851,-84.302,415.051,167.386,42.773,157.908
C06585=1029.844,-84.587,415.063,167.383,42.775,157.908
C06586=1029.838,-84.871,415.075,167.380,42.777,157.908
C06587=1029.830,-85.156,415.087,167.376,42.779,157.908
C06588=1029.824,-85.405,415.097,167.373,42.781,157.908
C06589=1029.819,-85.655,415.108,167.371,42.783,157.908
C06590=1029.812,-85.904,415.118,167.368,42.784,157.909
C06591=1029.807,-86.154,415.129,167.365,42.786,157.909
C06592=1029.801,-86.404,415.138,167.362,42.788,157.909
C06593=1029.794,-86.654,415.150,167.359,42.790,157.909
C06594=1029.788,-86.904,415.159,167.356,42.792,157.909
C06595=1029.782,-87.153,415.170,167.353,42.793,157.909
C06596=1029.777,-87.403,415.181,167.351,42.795,157.909
C06597=1029.770,-87.653,415.191,167.348,42.797,157.909
C06598=1029.765,-87.902,415.201,167.345,42.799,157.909
C06599=1029.758,-88.152,415.211,167.342,42.800,157.909
C06600=1029.753,-88.401,415.222,167.339,42.802,157.910
C06601=1029.746,-88.652,415.232,167.336,42.804,157.910
C06602=1029.740,-88.901,415.243,167.334,42.806,157.910
C06603=1029.734,-89.151,415.252,167.331,42.808,157.910
C06604=1029.728,-89.401,415.263,167.328,42.810,157.910
C06605=1029.722,-89.650,415.273,167.324,42.811,157.910
C06606=1029.716,-89.900,415.284,167.322,42.813,157.910
C06607=1029.711,-90.150,415.294,167.319,42.815,157.910
C06608=1029.704,-90.399,415.304,167.316,42.816,157.910
C06609=1029.699,-90.649,415.314,167.314,42.818,157.911
C06610=1029.693,-90.898,415.324,167.310,42.820,157.911
C06611=1029.687,-91.149,415.335,167.307,42.822,157.911
C06612=1029.681,-91.398,415.344,167.305,42.824,157.911
C06613=1029.675,-91.648,415.355,167.302,42.826,157.911
C06614=1029.669,-91.898,415.365,167.299,42.827,157.911
C06615=1029.663,-92.147,415.375,167.297,42.829,157.911
C06616=1029.657,-92.397,415.385,167.293,42.831,157.911
C06617=1029.652,-92.647,415.395,167.290,42.833,157.911
C06618=1029.645,-92.896,415.405,167.287,42.834,157.911
C06619=1029.640,-93.146,415.416,167.285,42.836,157.912
C06620=1029.633,-93.396,415.426,167.282,42.838,157.912
C06621=1029.628,-93.646,415.436,167.279,42.840,157.912
C06622=1029.622,-93.895,415.446,167.276,42.842,157.912
C06623=1029.616,-94.145,415.457,167.273,42.843,157.912
C06624=1029.610,-94.395,415.466,167.270,42.845,157.912
C06625=1029.604,-94.645,415.476,167.268,42.847,157.912
C06626=1029.599,-94.894,415.487,167.265,42.849,157.912
C06627=1029.592,-95.144,415.497,167.262,42.850,157.912
C06628=1029.587,-95.394,415.507,167.259,42.852,157.912
C06629=1029.581,-95.644,415.516,167.256,42.854,157.912
C06630=1029.575,-95.894,415.527,167.253,42.856,157.913
C06631=1029.570,-96.143,415.537,167.251,42.858,157.913
C06632=1029.564,-96.393,415.547,167.248,42.859,157.913
C06633=1029.558,-96.643,415.556,167.245,42.861,157.913
C06634=1029.551,-96.892,415.567,167.241,42.863,157.913
C06635=1029.546,-97.142,415.577,167.239,42.865,157.913
C06636=1029.540,-97.392,415.586,167.236,42.867,157.913
C06637=1029.534,-97.642,415.596,167.233,42.868,157.913
C06638=1029.528,-97.892,415.606,167.231,42.870,157.913
C06639=1029.522,-98.141,415.616,167.227,42.872,157.913
C06640=1029.516,-98.391,415.626,167.224,42.874,157.914
C06641=1029.511,-98.640,415.636,167.222,42.876,157.914
C06642=1029.505,-98.890,415.645,167.219,42.878,157.914
C06643=1029.498,-99.139,415.655,167.215,42.880,157.914
C06644=1029.493,-99.390,415.665,167.213,42.882,157.914
C06645=1029.487,-99.639,415.674,167.210,42.884,157.914
C06646=1029.481,-99.889,415.684,167.207,42.886,157.914
C06647=1029.474,-100.139,415.694,167.205,42.888,157.914
C06648=1029.468,-100.426,415.705,167.201,42.890,157.915
C06649=1029.462,-100.712,415.717,167.197,42.892,157.915
C06650=1029.455,-100.999,415.728,167.194,42.895,157.915
C06651=1029.447,-101.286,415.739,167.191,42.896,157.915
C06652=1029.442,-101.535,415.748,167.187,42.898,157.915
C06653=1029.436,-101.785,415.758,167.185,42.900,157.915
C06654=1029.430,-102.035,415.767,167.182,42.902,157.915
C06655=1029.424,-102.285,415.777,167.179,42.904,157.915
C06656=1029.418,-102.534,415.787,167.177,42.906,157.915
C06657=1029.412,-102.784,415.796,167.173,42.908,157.916
C06658=1029.406,-103.033,415.806,167.171,42.910,157.916
C06659=1029.401,-103.283,415.816,167.168,42.912,157.916
C06660=1029.395,-103.533,415.825,167.165,42.914,157.916
C06661=1029.389,-103.784,415.834,167.162,42.916,157.916
C06662=1029.383,-104.033,415.843,167.159,42.918,157.916
C06663=1029.377,-104.283,415.853,167.156,42.920,157.916
C06664=1029.371,-104.532,415.863,167.154,42.922,157.916
C06665=1029.365,-104.782,415.873,167.150,42.924,157.917
C06666=1029.360,-105.032,415.882,167.147,42.925,157.917
C06667=1029.354,-105.281,415.891,167.145,42.927,157.917
C06668=1029.347,-105.531,415.901,167.142,42.930,157.917
C06669=1029.341,-105.781,415.911,167.138,42.932,157.917
C06670=1029.336,-106.031,415.919,167.136,42.934,157.917
C06671=1029.331,-106.281,415.929,167.133,42.935,157.917
C06672=1029.324,-106.531,415.939,167.130,42.937,157.917
C06673=1029.319,-106.780,415.948,167.127,42.939,157.917
C06674=1029.313,-107.029,415.958,167.124,42.941,157.918
C06675=1029.307,-107.280,415.966,167.121,42.943,157.918
C06676=1029.301,-107.530,415.976,167.119,42.945,157.918
C06677=1029.295,-107.779,415.985,167.115,42.948,157.918
C06678=1029.289,-108.029,415.995,167.113,42.949,157.918
C06679=1029.283,-108.279,416.004,167.110,42.951,157.918
C06680=1029.277,-108.528,416.013,167.107,42.953,157.918
C06681=1029.271,-108.778,416.022,167.103,42.955,157.918
C06682=1029.265,-109.028,416.032,167.101,42.958,157.919
C06683=1029.260,-109.277,416.040,167.098,42.959,157.919
C06684=1029.254,-109.527,416.050,167.095,42.961,157.919
C06685=1029.248,-109.777,416.060,167.092,42.963,157.919
C06686=1029.242,-110.027,416.068,167.090,42.966,157.919
C06687=1029.236,-110.276,416.078,167.087,42.968,157.919
C06688=1029.230,-110.526,416.087,167.083,42.970,157.919
C06689=1029.225,-110.776,416.096,167.080,42.972,157.920
C06690=1029.219,-111.026,416.105,167.078,42.973,157.920
C06691=1029.212,-111.276,416.115,167.075,42.976,157.920
C06692=1029.207,-111.525,416.123,167.072,42.978,157.920
C06693=1029.201,-111.775,416.133,167.069,42.980,157.920
C06694=1029.196,-112.025,416.141,167.066,42.982,157.920
C06695=1029.189,-112.275,416.151,167.063,42.984,157.920
C06696=1029.183,-112.524,416.160,167.060,42.986,157.921
C06697=1029.178,-112.774,416.169,167.057,42.988,157.921
C06698=1029.172,-113.024,416.179,167.055,42.990,157.921
C06699=1029.167,-113.274,416.187,167.051,42.992,157.921
C06700=1029.160,-113.523,416.197,167.048,42.994,157.921
C06701=1029.155,-113.773,416.205,167.046,42.996,157.921
C06702=1029.149,-114.023,416.215,167.042,42.998,157.921
C06703=1029.143,-114.273,416.223,167.040,43.000,157.921
C06704=1029.138,-114.522,416.233,167.037,43.002,157.921
C06705=1029.132,-114.773,416.242,167.034,43.005,157.922
C06706=1029.125,-115.022,416.250,167.031,43.007,157.922
C06707=1029.120,-115.272,416.259,167.028,43.008,157.922
C06708=1029.114,-115.521,416.268,167.026,43.011,157.922
C06709=1029.108,-115.772,416.277,167.022,43.013,157.922
C06710=1029.102,-116.021,416.286,167.019,43.015,157.922
C06711=1029.097,-116.271,416.295,167.017,43.017,157.922
C06712=1029.090,-116.557,416.305,167.013,43.019,157.923
C06713=1029.083,-116.843,416.316,167.010,43.022,157.923
C06714=1029.077,-117.130,416.325,167.006,43.024,157.923
C06715=1029.070,-117.416,416.336,167.003,43.027,157.923
C06716=1029.065,-117.666,416.344,167.000,43.029,157.923
C06717=1029.058,-117.915,416.353,166.997,43.031,157.923
C06718=1029.052,-118.165,416.362,166.995,43.033,157.924
C06719=1029.047,-118.415,416.371,166.991,43.035,157.924
C06720=1029.041,-118.665,416.380,166.988,43.038,157.924
C06721=1029.035,-118.915,416.389,166.986,43.040,157.924
C06722=1029.029,-119.164,416.397,166.983,43.041,157.924
C06723=1029.024,-119.413,416.406,166.980,43.044,157.924
C06724=1029.018,-119.664,416.415,166.977,43.046,157.924
C06725=1029.012,-119.914,416.423,166.974,43.048,157.924
C06726=1029.006,-120.164,416.431,166.971,43.051,157.925
C06727=1029.000,-120.413,416.441,166.968,43.052,157.925
C06728=1028.994,-120.663,416.450,166.965,43.054,157.925
C06729=1028.989,-120.913,416.458,166.962,43.057,157.925
C06730=1028.984,-121.163,416.466,166.959,43.059,157.925
C06731=1028.977,-121.412,416.475,166.957,43.061,157.925
C06732=1028.972,-121.662,416.484,166.953,43.063,157.925
C06733=1028.966,-121.912,416.493,166.950,43.065,157.926
C06734=1028.960,-122.162,416.501,166.948,43.067,157.926
C06735=1028.954,-122.411,416.510,166.944,43.070,157.926
C06736=1028.948,-122.661,416.519,166.942,43.072,157.926
C06737=1028.943,-122.911,416.527,166.939,43.074,157.926
C06738=1028.936,-123.161,416.535,166.937,43.076,157.926
C06739=1028.931,-123.411,416.544,166.933,43.078,157.926
C06740=1028.926,-123.660,416.552,166.930,43.081,157.927
C06741=1028.920,-123.910,416.562,166.928,43.083,157.927
C06742=1028.914,-124.160,416.570,166.924,43.085,157.927
C06743=1028.908,-124.409,416.578,166.922,43.087,157.927
C06744=1028.903,-124.660,416.587,166.919,43.089,157.927
C06745=1028.897,-124.909,416.595,166.915,43.092,157.927
C06746=1028.891,-125.159,416.604,166.913,43.094,157.927
C06747=1028.885,-125.409,416.612,166.910,43.096,157.928
C06748=1028.879,-125.659,416.620,166.907,43.098,157.928
C06749=1028.874,-125.908,416.629,166.904,43.101,157.928
C06750=1028.868,-126.159,416.637,166.901,43.103,157.928
C06751=1028.862,-126.408,416.646,166.898,43.105,157.928
C06752=1028.856,-126.658,416.653,166.895,43.107,157.928
C06753=1028.850,-126.908,416.662,166.893,43.109,157.929
C06754=1028.844,-127.157,416.670,166.889,43.112,157.929
C06755=1028.839,-127.407,416.679,166.886,43.114,157.929
C06756=1028.833,-127.657,416.687,166.884,43.116,157.929
C06757=1028.828,-127.906,416.696,166.880,43.118,157.929
C06758=1028.822,-128.155,416.704,166.878,43.120,157.929
C06759=1028.818,-128.405,416.713,166.875,43.121,157.929
C06760=1028.814,-128.655,416.724,166.872,43.122,157.929
C06761=1028.810,-128.905,416.735,166.870,43.123,157.929
C06762=1028.808,-129.155,416.745,166.868,43.122,157.929
C06763=1028.805,-129.404,416.758,166.865,43.122,157.929
C06764=1028.803,-129.654,416.769,166.863,43.121,157.928
C06765=1028.803,-129.904,416.783,166.860,43.120,157.928
C06766=1028.802,-130.154,416.796,166.859,43.118,157.927
C06767=1028.802,-130.404,416.810,166.856,43.115,157.927
C06768=1028.803,-130.654,416.824,166.854,43.112,157.926
C06769=1028.805,-130.903,416.840,166.852,43.109,157.925
C06770=1028.806,-131.154,416.856,166.851,43.105,157.925
C06771=1028.810,-131.403,416.872,166.849,43.101,157.924
C06772=1028.813,-131.653,416.889,166.847,43.097,157.923
C06773=1028.816,-131.903,416.906,166.846,43.091,157.922
C06774=1028.821,-132.153,416.925,166.845,43.085,157.921
C06775=1028.826,-132.402,416.943,166.844,43.079,157.920
C06776=1028.512,-132.428,416.633,166.794,43.328,157.958
C06777=1028.506,-132.178,416.615,166.796,43.334,157.959
C06778=1028.502,-131.928,416.596,166.798,43.340,157.960
C06779=1028.498,-131.679,416.579,166.799,43.344,157.961
C06780=1028.496,-131.428,416.562,166.801,43.349,157.962
C06781=1028.492,-131.178,416.545,166.802,43.353,157.962
C06782=1028.490,-130.929,416.530,166.804,43.357,157.963
C06783=1028.489,-130.679,416.514,166.806,43.361,157.964
C06784=1028.488,-130.429,416.500,166.808,43.363,157.965
C06785=1028.488,-130.179,416.486,166.810,43.366,157.965
C06786=1028.488,-129.929,416.473,166.812,43.368,157.966
C06787=1028.489,-129.679,416.459,166.814,43.370,157.966
C06788=1028.491,-129.430,416.447,166.817,43.371,157.966
C06789=1028.493,-129.180,416.435,166.819,43.371,157.967
C06790=1028.496,-128.930,416.424,166.821,43.371,157.967
C06791=1028.499,-128.681,416.414,166.824,43.371,157.967
C06792=1028.503,-128.431,416.403,166.826,43.370,157.967
C06793=1028.508,-128.181,416.394,166.829,43.369,157.967
C06794=1028.513,-127.932,416.384,166.832,43.367,157.967
C06795=1028.519,-127.682,416.377,166.835,43.364,157.967
C06796=1028.524,-127.432,416.368,166.838,43.362,157.967
C06797=1028.530,-127.183,416.360,166.841,43.359,157.967
C06798=1028.536,-126.933,416.351,166.844,43.358,157.966
C06799=1028.542,-126.683,416.343,166.846,43.355,157.966
C06800=1028.547,-126.433,416.335,166.850,43.353,157.966
C06801=1028.554,-126.183,416.327,166.852,43.350,157.966
C06802=1028.559,-125.934,416.318,166.855,43.348,157.966
C06803=1028.564,-125.684,416.310,166.859,43.346,157.966
C06804=1028.570,-125.435,416.302,166.861,43.344,157.966
C06805=1028.576,-125.184,416.293,166.864,43.341,157.965
C06806=1028.582,-124.935,416.285,166.867,43.339,157.965
C06807=1028.587,-124.685,416.277,166.870,43.337,157.965
C06808=1028.593,-124.435,416.268,166.874,43.335,157.965
C06809=1028.599,-124.185,416.260,166.876,43.333,157.965
C06810=1028.605,-123.936,416.251,166.879,43.330,157.965
C06811=1028.611,-123.686,416.242,166.882,43.328,157.965
C06812=1028.617,-123.436,416.234,166.885,43.326,157.964
C06813=1028.622,-123.187,416.225,166.887,43.324,157.964
C06814=1028.628,-122.936,416.217,166.891,43.322,157.964
C06815=1028.633,-122.686,416.208,166.894,43.319,157.964
C06816=1028.640,-122.436,416.200,166.896,43.317,157.964
C06817=1028.645,-122.187,416.191,166.900,43.314,157.964
C06818=1028.650,-121.938,416.182,166.902,43.313,157.963
C06819=1028.657,-121.687,416.174,166.905,43.311,157.963
C06820=1028.662,-121.438,416.165,166.908,43.308,157.963
C06821=1028.667,-121.188,416.157,166.911,43.306,157.963
C06822=1028.674,-120.938,416.147,166.914,43.303,157.963
C06823=1028.680,-120.689,416.139,166.917,43.301,157.963
C06824=1028.686,-120.438,416.131,166.920,43.300,157.963
C06825=1028.691,-120.189,416.122,166.922,43.297,157.962
C06826=1028.697,-119.939,416.113,166.926,43.295,157.962
C06827=1028.702,-119.689,416.104,166.929,43.292,157.962
C06828=1028.708,-119.440,416.096,166.931,43.290,157.962
C06829=1028.714,-119.189,416.087,166.935,43.288,157.962
C06830=1028.720,-118.940,416.078,166.937,43.286,157.962
C06831=1028.726,-118.690,416.069,166.940,43.284,157.962
C06832=1028.732,-118.440,416.061,166.944,43.282,157.962
C06833=1028.738,-118.191,416.052,166.946,43.279,157.961
C06834=1028.743,-117.941,416.043,166.949,43.278,157.961
C06835=1028.749,-117.690,416.034,166.952,43.275,157.961
C06836=1028.754,-117.441,416.025,166.955,43.273,157.961
C06837=1028.762,-117.154,416.016,166.958,43.270,157.961
C06838=1028.768,-116.869,416.005,166.962,43.268,157.961
C06839=1028.775,-116.583,415.995,166.965,43.266,157.960
C06840=1028.781,-116.296,415.985,166.968,43.263,157.960
C06841=1028.787,-116.047,415.977,166.972,43.261,157.960
C06842=1028.793,-115.797,415.968,166.974,43.259,157.960
C06843=1028.799,-115.547,415.958,166.977,43.256,157.960
C06844=1028.805,-115.297,415.950,166.980,43.254,157.960
C06845=1028.810,-115.048,415.940,166.983,43.252,157.960
C06846=1028.816,-114.797,415.932,166.986,43.250,157.959
C06847=1028.822,-114.548,415.922,166.988,43.248,157.959
C06848=1028.828,-114.298,415.914,166.992,43.246,157.959
C06849=1028.834,-114.049,415.905,166.994,43.243,157.959
C06850=1028.840,-113.799,415.896,166.997,43.242,157.959
C06851=1028.846,-113.549,415.887,167.001,43.240,157.959
C06852=1028.851,-113.299,415.878,167.003,43.238,157.959
C06853=1028.857,-113.049,415.868,167.006,43.235,157.959
C06854=1028.862,-112.800,415.860,167.010,43.233,157.958
C06855=1028.869,-112.550,415.850,167.012,43.231,157.958
C06856=1028.874,-112.300,415.842,167.015,43.229,157.958
C06857=1028.880,-112.050,415.832,167.018,43.227,157.958
C06858=1028.886,-111.800,415.824,167.021,43.225,157.958
C06859=1028.891,-111.551,415.814,167.024,43.223,157.958
C06860=1028.898,-111.301,415.805,167.026,43.221,157.958
C06861=1028.903,-111.051,415.796,167.030,43.218,157.958
C06862=1028.909,-110.802,415.787,167.033,43.216,157.957
C06863=1028.915,-110.552,415.777,167.035,43.214,157.957
C06864=1028.921,-110.302,415.769,167.039,43.212,157.957
C06865=1028.927,-110.052,415.759,167.041,43.210,157.957
C06866=1028.933,-109.802,415.750,167.044,43.208,157.957
C06867=1028.938,-109.553,415.741,167.048,43.206,157.957
C06868=1028.944,-109.303,415.731,167.050,43.203,157.957
C06869=1028.950,-109.053,415.723,167.053,43.202,157.956
C06870=1028.956,-108.803,415.713,167.055,43.200,157.956
C06871=1028.962,-108.554,415.704,167.059,43.198,157.956
C06872=1028.968,-108.304,415.694,167.062,43.195,157.956
C06873=1028.973,-108.054,415.686,167.064,43.193,157.956
C06874=1028.980,-107.804,415.676,167.068,43.191,157.956
C06875=1028.986,-107.555,415.667,167.071,43.189,157.956
C06876=1028.991,-107.305,415.658,167.073,43.187,157.956
C06877=1028.997,-107.055,415.649,167.077,43.185,157.955
C06878=1029.003,-106.805,415.639,167.079,43.183,157.955
C06879=1029.008,-106.556,415.629,167.082,43.181,157.955
C06880=1029.014,-106.306,415.620,167.085,43.179,157.955
C06881=1029.020,-106.056,415.611,167.088,43.177,157.955
C06882=1029.026,-105.806,415.601,167.091,43.175,157.955
C06883=1029.032,-105.557,415.592,167.094,43.173,157.955
C06884=1029.038,-105.307,415.582,167.096,43.171,157.955
C06885=1029.044,-105.057,415.573,167.100,43.169,157.955
C06886=1029.049,-104.808,415.563,167.103,43.167,157.954
C06887=1029.055,-104.558,415.554,167.105,43.165,157.954
C06888=1029.061,-104.308,415.545,167.109,43.163,157.954
C06889=1029.067,-104.058,415.535,167.111,43.161,157.954
C06890=1029.073,-103.809,415.526,167.114,43.159,157.954
C06891=1029.079,-103.559,415.516,167.117,43.157,157.954
C06892=1029.084,-103.309,415.506,167.120,43.155,157.954
C06893=1029.091,-103.059,415.497,167.123,43.153,157.954
C06894=1029.096,-102.810,415.487,167.126,43.151,157.953
C06895=1029.102,-102.560,415.478,167.128,43.149,157.953
C06896=1029.108,-102.310,415.468,167.132,43.146,157.953
C06897=1029.114,-102.060,415.458,167.134,43.145,157.953
C06898=1029.120,-101.810,415.449,167.137,43.143,157.953
C06899=1029.126,-101.561,415.439,167.140,43.141,157.953
C06900=1029.132,-101.311,415.430,167.143,43.139,157.953
C06901=1029.139,-101.025,415.419,167.146,43.137,157.953
C06902=1029.145,-100.737,415.407,167.150,43.134,157.952
C06903=1029.152,-100.451,415.396,167.153,43.132,157.952
C06904=1029.159,-100.164,415.385,167.157,43.130,157.952
C06905=1029.165,-99.914,415.376,167.159,43.128,157.952
C06906=1029.171,-99.664,415.366,167.162,43.126,157.952
C06907=1029.177,-99.415,415.357,167.166,43.124,157.952
C06908=1029.182,-99.165,415.347,167.168,43.122,157.952
C06909=1029.188,-98.916,415.337,167.171,43.120,157.952
C06910=1029.195,-98.666,415.327,167.174,43.118,157.951
C06911=1029.201,-98.416,415.317,167.177,43.116,157.951
C06912=1029.206,-98.166,415.307,167.180,43.114,157.951
C06913=1029.212,-97.917,415.298,167.183,43.112,157.951
C06914=1029.219,-97.667,415.288,167.185,43.110,157.951
C06915=1029.224,-97.417,415.278,167.189,43.108,157.951
C06916=1029.230,-97.168,415.269,167.192,43.106,157.951
C06917=1029.235,-96.918,415.258,167.194,43.104,157.951
C06918=1029.241,-96.668,415.248,167.197,43.102,157.951
C06919=1029.247,-96.418,415.238,167.200,43.100,157.950
C06920=1029.253,-96.168,415.229,167.203,43.098,157.950
C06921=1029.259,-95.919,415.218,167.206,43.097,157.950
C06922=1029.265,-95.669,415.208,167.209,43.095,157.950
C06923=1029.270,-95.419,415.198,167.211,43.093,157.950
C06924=1029.277,-95.169,415.188,167.214,43.091,157.950
C06925=1029.282,-94.920,415.178,167.218,43.090,157.950
C06926=1029.288,-94.671,415.168,167.220,43.088,157.950
C06927=1029.293,-94.420,415.158,167.223,43.086,157.950
C06928=1029.300,-94.171,415.148,167.226,43.084,157.950
C06929=1029.305,-93.921,415.138,167.228,43.082,157.950
C06930=1029.311,-93.671,415.128,167.232,43.080,157.949
C06931=1029.317,-93.421,415.118,167.235,43.078,157.949
C06932=1029.323,-93.172,415.108,167.237,43.077,157.949
C06933=1029.329,-92.922,415.098,167.240,43.075,157.949
C06934=1029.335,-92.673,415.087,167.243,43.073,157.949
C06935=1029.341,-92.423,415.077,167.246,43.071,157.949
C06936=1029.347,-92.173,415.068,167.249,43.069,157.949
C06937=1029.353,-91.923,415.057,167.252,43.067,157.949
C06938=1029.359,-91.674,415.047,167.254,43.065,157.949
C06939=1029.364,-91.423,415.037,167.257,43.063,157.948
C06940=1029.371,-91.174,415.027,167.261,43.061,157.948
C06941=1029.376,-90.924,415.017,167.263,43.060,157.948
C06942=1029.383,-90.675,415.006,167.266,43.058,157.948
C06943=1029.388,-90.425,414.996,167.269,43.056,157.948
C06944=1029.394,-90.176,414.986,167.272,43.055,157.948
C06945=1029.400,-89.926,414.976,167.275,43.053,157.948
C06946=1029.406,-89.676,414.966,167.278,43.051,157.948
C06947=1029.412,-89.426,414.955,167.281,43.049,157.948
C06948=1029.417,-89.176,414.945,167.283,43.047,157.948
C06949=1029.424,-88.927,414.935,167.286,43.045,157.948
C06950=1029.430,-88.676,414.924,167.289,43.043,157.947
C06951=1029.436,-88.427,414.914,167.292,43.041,157.947
C06952=1029.442,-88.177,414.904,167.295,43.040,157.947
C06953=1029.448,-87.928,414.893,167.298,43.038,157.947
C06954=1029.454,-87.678,414.883,167.300,43.036,157.947
C06955=1029.460,-87.428,414.873,167.303,43.034,157.947
C06956=1029.466,-87.179,414.862,167.307,43.032,157.947
C06957=1029.471,-86.929,414.852,167.309,43.030,157.947
C06958=1029.478,-86.680,414.842,167.312,43.028,157.947
C06959=1029.483,-86.430,414.832,167.315,43.026,157.946
C06960=1029.490,-86.180,414.821,167.317,43.025,157.946
C06961=1029.496,-85.930,414.811,167.321,43.023,157.946
C06962=1029.502,-85.680,414.800,167.324,43.021,157.946
C06963=1029.508,-85.431,414.790,167.326,43.019,157.946
C06964=1029.514,-85.181,414.780,167.329,43.017,157.946
C06965=1029.521,-84.896,414.768,167.333,43.015,157.946
C06966=1029.528,-84.612,414.756,167.335,43.013,157.946
C06967=1029.535,-84.328,414.744,167.339,43.011,157.946
C06968=1029.541,-84.043,414.732,167.343,43.009,157.946
C06969=1029.547,-83.793,414.722,167.345,43.007,157.945
C06970=1029.553,-83.544,414.711,167.348,43.005,157.945
C06971=1029.560,-83.294,414.700,167.351,43.004,157.945
C06972=1029.566,-83.044,414.690,167.354,43.002,157.945
C06973=1029.571,-82.794,414.679,167.357,43.000,157.945
C06974=1029.578,-82.545,414.669,167.360,42.998,157.945
C06975=1029.584,-82.296,414.658,167.362,42.996,157.945
C06976=1029.590,-82.045,414.648,167.365,42.994,157.945
C06977=1029.596,-81.796,414.637,167.368,42.992,157.945
C06978=1029.602,-81.546,414.627,167.371,42.990,157.944
C06979=1029.608,-81.296,414.617,167.374,42.989,157.944
C06980=1029.614,-81.046,414.606,167.377,42.987,157.944
C06981=1029.621,-80.797,414.596,167.379,42.985,157.944
C06982=1029.627,-80.548,414.585,167.382,42.983,157.944
C06983=1029.632,-80.297,414.574,167.386,42.981,157.944
C06984=1029.639,-80.048,414.564,167.388,42.979,157.944
C06985=1029.645,-79.798,414.553,167.391,42.977,157.944
C06986=1029.651,-79.549,414.542,167.394,42.976,157.944
C06987=1029.657,-79.298,414.531,167.397,42.974,157.944
C06988=1029.663,-79.049,414.520,167.399,42.972,157.943
C06989=1029.669,-78.800,414.510,167.402,42.971,157.943
C06990=1029.675,-78.550,414.499,167.406,42.969,157.943
C06991=1029.681,-78.299,414.488,167.408,42.967,157.943
C06992=1029.687,-78.050,414.477,167.411,42.966,157.943
C06993=1029.692,-77.800,414.467,167.414,42.964,157.943
C06994=1029.699,-77.550,414.455,167.416,42.962,157.943
C06995=1029.705,-77.301,414.445,167.419,42.960,157.943
C06996=1029.711,-77.052,414.434,167.422,42.959,157.943
C06997=1029.717,-76.802,414.423,167.425,42.957,157.943
C06998=1029.723,-76.552,414.412,167.428,42.955,157.943
C06999=1029.729,-76.302,414.401,167.431,42.953,157.942
C07000=1029.735,-76.053,414.390,167.434,42.952,157.942
C07001=1029.741,-75.803,414.379,167.437,42.950,157.942
C07002=1029.747,-75.553,414.368,167.439,42.948,157.942
C07003=1029.753,-75.304,414.358,167.442,42.947,157.942
C07004=1029.759,-75.054,414.347,167.445,42.945,157.942
C07005=1029.765,-74.804,414.336,167.447,42.944,157.942
C07006=1029.772,-74.554,414.324,167.451,42.942,157.942
C07007=1029.777,-74.305,414.314,167.454,42.940,157.942
C07008=1029.783,-74.055,414.303,167.456,42.938,157.942
C07009=1029.789,-73.805,414.291,167.459,42.937,157.942
C07010=1029.795,-73.556,414.280,167.462,42.935,157.942
C07011=1029.801,-73.307,414.269,167.465,42.933,157.941
C07012=1029.807,-73.056,414.257,167.467,42.932,157.941
C07013=1029.812,-72.807,414.246,167.470,42.930,157.941
C07014=1029.818,-72.557,414.235,167.473,42.929,157.941
C07015=1029.825,-72.307,414.224,167.476,42.927,157.941
C07016=1029.831,-72.058,414.213,167.478,42.925,157.941
C07017=1029.836,-71.809,414.202,167.481,42.924,157.941
C07018=1029.843,-71.558,414.190,167.484,42.922,157.941
C07019=1029.848,-71.309,414.179,167.487,42.921,157.941
C07020=1029.854,-71.059,414.167,167.489,42.919,157.941
C07021=1029.860,-70.810,414.156,167.492,42.917,157.941
C07022=1029.866,-70.560,414.145,167.495,42.916,157.941
C07023=1029.872,-70.310,414.134,167.499,42.914,157.941
C07024=1029.878,-70.061,414.122,167.501,42.913,157.941
C07025=1029.884,-69.811,414.111,167.504,42.911,157.941
C07026=1029.890,-69.561,414.100,167.507,42.909,157.940
C07027=1029.896,-69.311,414.088,167.510,42.908,157.940
C07028=1029.902,-69.062,414.077,167.512,42.906,157.940
C07029=1029.909,-68.779,414.064,167.515,42.905,157.940
C07030=1029.915,-68.497,414.051,167.519,42.903,157.940
C07031=1029.922,-68.215,414.039,167.522,42.901,157.940
C07032=1029.929,-67.932,414.026,167.525,42.899,157.940
C07033=1029.935,-67.683,414.014,167.528,42.898,157.940
C07034=1029.941,-67.433,414.002,167.531,42.896,157.940
C07035=1029.946,-67.183,413.992,167.533,42.895,157.940
C07036=1029.953,-66.934,413.980,167.536,42.893,157.940
C07037=1029.959,-66.684,413.969,167.539,42.892,157.940
C07038=1029.965,-66.435,413.957,167.542,42.890,157.940
C07039=1029.970,-66.185,413.945,167.544,42.888,157.939
C07040=1029.977,-65.935,413.934,167.547,42.887,157.939
C07041=1029.983,-65.686,413.922,167.550,42.885,157.939
C07042=1029.989,-65.436,413.911,167.553,42.884,157.939
C07043=1029.995,-65.187,413.900,167.555,42.882,157.939
C07044=1030.001,-64.936,413.888,167.558,42.880,157.939
C07045=1030.007,-64.687,413.876,167.561,42.879,157.939
C07046=1030.013,-64.437,413.865,167.563,42.877,157.939
C07047=1030.020,-64.187,413.854,167.566,42.875,157.939
C07048=1030.026,-63.938,413.842,167.569,42.874,157.939
C07049=1030.031,-63.688,413.830,167.572,42.872,157.939
C07050=1030.037,-63.439,413.819,167.575,42.871,157.939
C07051=1030.044,-63.189,413.807,167.577,42.869,157.939
C07052=1030.050,-62.939,413.795,167.580,42.867,157.938
C07053=1030.056,-62.690,413.785,167.583,42.866,157.938
C07054=1030.062,-62.440,413.772,167.585,42.864,157.938
C07055=1030.068,-62.191,413.760,167.589,42.862,157.938
C07056=1030.074,-61.941,413.749,167.592,42.861,157.938
C07057=1030.081,-61.691,413.737,167.595,42.859,157.938
C07058=1030.086,-61.441,413.726,167.597,42.858,157.938
C07059=1030.093,-61.192,413.714,167.600,42.856,157.938
C07060=1030.098,-60.942,413.703,167.603,42.855,157.938
C07061=1030.105,-60.693,413.691,167.606,42.854,157.938
C07062=1030.111,-60.442,413.679,167.608,42.852,157.938
C07063=1030.117,-60.193,413.668,167.611,42.850,157.938
C07064=1030.123,-59.944,413.656,167.614,42.849,157.938
C07065=1030.130,-59.694,413.644,167.617,42.847,157.938
C07066=1030.136,-59.445,413.633,167.619,42.845,157.937
C07067=1030.142,-59.195,413.620,167.622,42.844,157.937
C07068=1030.148,-58.945,413.609,167.625,42.842,157.937
C07069=1030.154,-58.696,413.597,167.627,42.840,157.937
C07070=1030.161,-58.446,413.585,167.630,42.839,157.937
C07071=1030.166,-58.196,413.574,167.633,42.837,157.937
C07072=1030.172,-57.947,413.562,167.636,42.835,157.937
C07073=1030.179,-57.697,413.550,167.638,42.834,157.937
C07074=1030.185,-57.447,413.539,167.641,42.832,157.937
C07075=1030.191,-57.197,413.526,167.644,42.831,157.937
C07076=1030.197,-56.948,413.515,167.647,42.829,157.937
C07077=1030.203,-56.698,413.503,167.649,42.828,157.937
C07078=1030.210,-56.449,413.491,167.652,42.826,157.936
C07079=1030.216,-56.199,413.479,167.655,42.825,157.936
C07080=1030.222,-55.950,413.467,167.657,42.823,157.936
C07081=1030.228,-55.700,413.456,167.660,42.821,157.936
C07082=1030.234,-55.450,413.443,167.663,42.820,157.936
C07083=1030.241,-55.200,413.431,167.666,42.818,157.936
C07084=1030.247,-54.951,413.420,167.668,42.816,157.936
C07085=1030.253,-54.701,413.409,167.671,42.815,157.936
C07086=1030.259,-54.451,413.396,167.674,42.813,157.936
C07087=1030.266,-54.202,413.384,167.677,42.811,157.936
C07088=1030.272,-53.953,413.373,167.679,42.810,157.936
C07089=1030.279,-53.703,413.361,167.682,42.808,157.936
C07090=1030.284,-53.453,413.349,167.685,42.807,157.935
C07091=1030.291,-53.203,413.337,167.689,42.805,157.935
C07092=1030.298,-52.954,413.325,167.691,42.803,157.935
C07093=1030.304,-52.672,413.311,167.694,42.802,157.935
C07094=1030.311,-52.392,413.298,167.697,42.800,157.935
C07095=1030.318,-52.110,413.285,167.700,42.798,157.935
C07096=1030.326,-51.829,413.271,167.703,42.796,157.935
C07097=1030.332,-51.579,413.258,167.706,42.795,157.935
C07098=1030.338,-51.331,413.247,167.708,42.793,157.935
C07099=1030.345,-51.081,413.235,167.711,42.791,157.935
C07100=1030.350,-50.831,413.223,167.714,42.790,157.935
C07101=1030.357,-50.581,413.211,167.717,42.788,157.934
C07102=1030.363,-50.331,413.198,167.720,42.787,157.935
C07103=1030.369,-50.081,413.186,167.722,42.785,157.934
C07104=1030.375,-49.832,413.174,167.725,42.784,157.934
C07105=1030.381,-49.582,413.161,167.728,42.782,157.934
C07106=1030.387,-49.333,413.150,167.731,42.781,157.934
C07107=1030.393,-49.083,413.137,167.733,42.780,157.934
C07108=1030.399,-48.834,413.124,167.736,42.778,157.934
C07109=1030.406,-48.584,413.112,167.739,42.777,157.934
C07110=1030.412,-48.334,413.099,167.742,42.775,157.934
C07111=1030.418,-48.084,413.087,167.743,42.774,157.934
C07112=1030.424,-47.836,413.075,167.746,42.772,157.934
C07113=1030.430,-47.586,413.063,167.749,42.771,157.934
C07114=1030.436,-47.336,413.050,167.752,42.769,157.934
C07115=1030.442,-47.086,413.038,167.755,42.768,157.934
C07116=1030.448,-46.836,413.026,167.757,42.767,157.934
C07117=1030.454,-46.587,413.012,167.760,42.765,157.934
C07118=1030.461,-46.337,413.000,167.763,42.764,157.934
C07119=1030.467,-46.088,412.988,167.766,42.762,157.933
C07120=1030.473,-45.838,412.975,167.768,42.761,157.933
C07121=1030.480,-45.588,412.963,167.771,42.759,157.933
C07122=1030.485,-45.340,412.950,167.774,42.758,157.933
C07123=1030.491,-45.090,412.938,167.776,42.757,157.933
C07124=1030.498,-44.840,412.926,167.779,42.755,157.933
C07125=1030.504,-44.590,412.913,167.781,42.754,157.933
C07126=1030.510,-44.340,412.901,167.784,42.752,157.933
C07127=1030.517,-44.091,412.888,167.787,42.751,157.933
C07128=1030.522,-43.841,412.876,167.790,42.750,157.933
C07129=1030.528,-43.592,412.863,167.792,42.748,157.933
C07130=1030.534,-43.342,412.850,167.795,42.747,157.933
C07131=1030.541,-43.093,412.838,167.798,42.745,157.933
C07132=1030.547,-42.843,412.825,167.801,42.744,157.933
C07133=1030.553,-42.593,412.813,167.803,42.742,157.933
C07134=1030.560,-42.343,412.801,167.806,42.741,157.933
C07135=1030.566,-42.094,412.787,167.808,42.740,157.932
C07136=1030.572,-41.844,412.775,167.811,42.738,157.932
C07137=1030.578,-41.595,412.763,167.814,42.737,157.932
C07138=1030.585,-41.345,412.750,167.816,42.735,157.932
C07139=1030.591,-41.096,412.737,167.819,42.734,157.932
C07140=1030.596,-40.846,412.725,167.822,42.732,157.932
C07141=1030.603,-40.597,412.712,167.825,42.731,157.932
C07142=1030.609,-40.347,412.699,167.827,42.729,157.932
C07143=1030.615,-40.097,412.687,167.830,42.728,157.932
C07144=1030.622,-39.848,412.674,167.833,42.727,157.932
C07145=1030.628,-39.598,412.662,167.836,42.725,157.932
C07146=1030.634,-39.349,412.648,167.837,42.724,157.932
C07147=1030.640,-39.099,412.636,167.840,42.722,157.932
C07148=1030.647,-38.849,412.624,167.843,42.721,157.932
C07149=1030.653,-38.600,412.610,167.846,42.719,157.932
C07150=1030.660,-38.350,412.598,167.849,42.718,157.932
C07151=1030.666,-38.100,412.584,167.851,42.717,157.932
C07152=1030.672,-37.850,412.572,167.854,42.715,157.931
C07153=1030.678,-37.601,412.558,167.856,42.714,157.931
C07154=1030.684,-37.351,412.546,167.859,42.713,157.931
C07155=1030.690,-37.102,412.533,167.861,42.711,157.931
C07156=1030.696,-36.852,412.520,167.864,42.710,157.931
C07157=1030.703,-36.572,412.505,167.867,42.709,157.931
C07158=1030.710,-36.291,412.491,167.870,42.707,157.931
C07159=1030.717,-36.010,412.476,167.874,42.706,157.931
C07160=1030.723,-35.730,412.461,167.876,42.704,157.931
C07161=1030.730,-35.480,412.448,167.879,42.703,157.931
C07162=1030.736,-35.230,412.436,167.881,42.701,157.931
C07163=1030.742,-34.981,412.422,167.884,42.700,157.931
C07164=1030.748,-34.732,412.409,167.887,42.699,157.931
C07165=1030.754,-34.482,412.397,167.889,42.697,157.931
C07166=1030.761,-34.232,412.383,167.892,42.696,157.931
C07167=1030.767,-33.982,412.370,167.895,42.695,157.931
C07168=1030.773,-33.733,412.357,167.897,42.693,157.930
C07169=1030.779,-33.484,412.344,167.899,42.692,157.930
C07170=1030.785,-33.234,412.331,167.902,42.691,157.930
C07171=1030.791,-32.984,412.318,167.905,42.689,157.930
C07172=1030.797,-32.735,412.305,167.908,42.688,157.930
C07173=1030.804,-32.485,412.292,167.911,42.686,157.930
C07174=1030.810,-32.235,412.279,167.912,42.685,157.930
C07175=1030.816,-31.986,412.265,167.915,42.684,157.930
C07176=1030.822,-31.736,412.253,167.918,42.682,157.930
C07177=1030.829,-31.487,412.240,167.921,42.681,157.930
C07178=1030.835,-31.238,412.227,167.924,42.680,157.930
C07179=1030.842,-30.988,412.213,167.926,42.678,157.930
C07180=1030.847,-30.738,412.200,167.928,42.677,157.930
C07181=1030.854,-30.489,412.187,167.931,42.675,157.930
C07182=1030.860,-30.239,412.173,167.934,42.674,157.930
C07183=1030.867,-29.989,412.160,167.937,42.673,157.930
C07184=1030.873,-29.739,412.147,167.939,42.671,157.930
C07185=1030.879,-29.490,412.134,167.942,42.670,157.930
C07186=1030.885,-29.241,412.121,167.944,42.669,157.930
C07187=1030.891,-28.992,412.107,167.947,42.667,157.929
C07188=1030.898,-28.741,412.095,167.949,42.666,157.929
C07189=1030.904,-28.492,412.081,167.952,42.664,157.929
C07190=1030.910,-28.243,412.068,167.955,42.663,157.929
C07191=1030.916,-27.993,412.055,167.958,42.662,157.929
C07192=1030.923,-27.743,412.041,167.959,42.660,157.929
C07193=1030.929,-27.493,412.029,167.962,42.659,157.929
C07194=1030.935,-27.244,412.015,167.965,42.657,157.929
C07195=1030.942,-26.994,412.002,167.968,42.656,157.929
C07196=1030.948,-26.745,411.988,167.971,42.655,157.929
C07197=1030.954,-26.495,411.974,167.973,42.654,157.929
C07198=1030.960,-26.246,411.961,167.975,42.652,157.929
C07199=1030.967,-25.996,411.948,167.978,42.651,157.929
C07200=1030.973,-25.747,411.934,167.981,42.650,157.929
C07201=1030.979,-25.497,411.920,167.983,42.649,157.929
C07202=1030.985,-25.248,411.907,167.986,42.648,157.929
C07203=1030.992,-24.998,411.894,167.988,42.646,157.929
C07204=1030.998,-24.749,411.880,167.991,42.645,157.929
C07205=1031.003,-24.499,411.866,167.993,42.644,157.929
C07206=1031.010,-24.249,411.853,167.996,42.643,157.929
C07207=1031.016,-24.000,411.839,167.999,42.641,157.928
C07208=1031.022,-23.750,411.826,168.001,42.640,157.928
C07209=1031.029,-23.500,411.812,168.003,42.639,157.928
C07210=1031.035,-23.251,411.799,168.006,42.638,157.928
C07211=1031.041,-23.002,411.785,168.009,42.636,157.928
C07212=1031.047,-22.752,411.771,168.012,42.635,157.928
C07213=1031.053,-22.502,411.758,168.014,42.634,157.928
C07214=1031.060,-22.253,411.745,168.016,42.633,157.928
C07215=1031.066,-22.003,411.730,168.019,42.631,157.928
C07216=1031.072,-21.754,411.717,168.022,42.630,157.928
C07217=1031.078,-21.504,411.704,168.025,42.629,157.928
C07218=1031.084,-21.254,411.690,168.026,42.627,157.928
C07219=1031.091,-21.005,411.676,168.029,42.626,157.928
C07220=1031.097,-20.756,411.662,168.032,42.625,157.928
C07221=1031.104,-20.474,411.647,168.035,42.623,157.928
C07222=1031.111,-20.193,411.631,168.038,42.622,157.928
C07223=1031.118,-19.911,411.616,168.040,42.621,157.928
C07224=1031.125,-19.630,411.601,168.043,42.619,157.928
C07225=1031.131,-19.380,411.587,168.046,42.618,157.928
C07226=1031.138,-19.130,411.574,168.049,42.617,157.928
C07227=1031.145,-18.881,411.559,168.051,42.615,157.927
C07228=1031.150,-18.632,411.545,168.053,42.614,157.927
C07229=1031.156,-18.382,411.532,168.056,42.613,157.927
C07230=1031.163,-18.132,411.519,168.059,42.611,157.927
C07231=1031.169,-17.883,411.505,168.061,42.610,157.927
C07232=1031.176,-17.633,411.490,168.064,42.609,157.927
C07233=1031.182,-17.384,411.477,168.066,42.608,157.927
C07234=1031.188,-17.134,411.463,168.069,42.606,157.927
C07235=1031.194,-16.885,411.450,168.071,42.605,157.927
C07236=1031.200,-16.635,411.436,168.074,42.604,157.927
C07237=1031.207,-16.386,411.421,168.077,42.602,157.927
C07238=1031.213,-16.136,411.408,168.079,42.601,157.927
C07239=1031.220,-15.886,411.394,168.081,42.600,157.927
C07240=1031.226,-15.638,411.380,168.084,42.598,157.927
C07241=1031.232,-15.388,411.366,168.087,42.597,157.927
C07242=1031.238,-15.138,411.352,168.090,42.596,157.927
C07243=1031.245,-14.889,411.338,168.091,42.595,157.927
C07244=1031.251,-14.639,411.324,168.094,42.594,157.927
C07245=1031.257,-14.389,411.310,168.097,42.592,157.927
C07246=1031.263,-14.140,411.296,168.099,42.591,157.926
C07247=1031.269,-13.890,411.282,168.102,42.590,157.926
C07248=1031.275,-13.641,411.268,168.105,42.589,157.926
C07249=1031.282,-13.391,411.253,168.106,42.588,157.926
C07250=1031.288,-13.142,411.240,168.109,42.586,157.926
C07251=1031.294,-12.892,411.225,168.112,42.585,157.926
C07252=1031.300,-12.642,411.211,168.114,42.584,157.926
C07253=1031.307,-12.393,411.197,168.117,42.583,157.926
C07254=1031.313,-12.144,411.183,168.119,42.581,157.926
C07255=1031.319,-11.894,411.170,168.121,42.580,157.926
C07256=1031.325,-11.645,411.155,168.124,42.579,157.926
C07257=1031.332,-11.395,411.141,168.127,42.578,157.926
C07258=1031.338,-11.146,411.127,168.130,42.576,157.926
C07259=1031.344,-10.895,411.112,168.132,42.575,157.926
C07260=1031.350,-10.647,411.099,168.134,42.574,157.926
C07261=1031.356,-10.396,411.084,168.137,42.573,157.926
C07262=1031.363,-10.148,411.070,168.139,42.572,157.926
C07263=1031.369,-9.898,411.056,168.142,42.570,157.926
C07264=1031.375,-9.648,411.041,168.145,42.569,157.926
C07265=1031.382,-9.399,411.028,168.146,42.568,157.926
C07266=1031.388,-9.149,411.013,168.149,42.567,157.926
C07267=1031.394,-8.900,410.998,168.152,42.566,157.926
C07268=1031.401,-8.650,410.985,168.154,42.564,157.925
C07269=1031.406,-8.401,410.970,168.157,42.563,157.925
C07270=1031.413,-8.151,410.956,168.160,42.562,157.925
C07271=1031.420,-7.901,410.942,168.161,42.561,157.925
C07272=1031.425,-7.652,410.928,168.164,42.559,157.925
C07273=1031.432,-7.403,410.913,168.167,42.558,157.925
C07274=1031.438,-7.154,410.899,168.169,42.557,157.925
C07275=1031.445,-6.904,410.885,168.172,42.556,157.925
C07276=1031.451,-6.654,410.870,168.175,42.555,157.925
C07277=1031.457,-6.404,410.856,168.176,42.553,157.925
C07278=1031.464,-6.155,410.842,168.179,42.552,157.925
C07279=1031.470,-5.905,410.827,168.182,42.551,157.925
C07280=1031.476,-5.656,410.813,168.184,42.550,157.925
